Omron CX-Programmer project NewProject (CX-Programmer 9.66)

# PLC NewPLC1: CP1H XA

## Global symbols (name address type ; comment)
AI_SAW_CURRENT 200 CHANNEL  ; ANALOG.INPUT1.SAW.CURRENT
AI_TRANS_AXIS_DRIVE_VEL_FDBK 201 CHANNEL  ; AI.TRANSVERSE.AXIS.DRIVE.VELOCITY.FEEDBACK
AO_TRANS_VEL_REF 210 CHANNEL  ; TRANSVERSE.AXIS.VELOCITY.ANALOG.REFERENCE
0.05 BOOL  ; SPARE - Possible Zone Interference Limit Switch Input.
1024 CHANNEL  ; Encoder PPR
1.03 BOOL  ; Spare
200 CHANNEL  ; Saw Motor Current Input
210 CHANNEL  ; Cross Travel Speed Refernce Command
40 CHANNEL  ; OI.SCALING.SAW.CURRENT.PART1
8.00 BOOL  ; Place holder for Automatic PID control request
A434.04 BOOL  ; Analog IO Initialised
D100 CHANNEL  ; M_BLOCK_HEIGHT_INT_RAW
D10000 CHANNEL  ; OPERATION.PROGRAM.CHECK.BLOCK1.BLOCK.HEIGHT
D10001 CHANNEL  ; OPERATION.CHECK.PROGRAM.BLOCK1.BLOCK.QUANTITY
D10002 CHANNEL  ; OPERATION.PROGRAM.CHECK.BLOCK1.FORWARD.POSITION
D10003 CHANNEL  ; OPERATION.PROGRAM.CHECK.BLOCK1.FIRST.CUT
D10004 CHANNEL  ; OPERATION.PROGRAM.CHECK.BLOCK1.NUMBER.OF.SLABS
D10006 CHANNEL  ; OPERATION.PROGRAM.CHECK.BLOCK1.SLAB1.QUANTITY
D10007 CHANNEL  ; OPERATION.PROGRAM.CHECK.BLOCK1.SLAB2.SIZE
D10008 CHANNEL  ; OPERATION.PROGRAM.CHECK.BLOCK1.SLAB2.QUANTITY
D10009 CHANNEL  ; OPERATION.PROGRAM.CHECK.BLOCK1.SLAB3.SIZE
D1001 CHANNEL  ; Block 1 Data - Number of Blocks
D10010 CHANNEL  ; OPERATION.PROGRAM.CHECK.BLOCK1.SLAB1.SIZE
D10010 CHANNEL  ; OPERATION.PROGRAM.CHECK.BLOCK1.SLAB1.SIZE
D10011 CHANNEL  ; OPERATION.PROGRAM.CHECK.BLOCK1.SLAB4.SIZE
D10012 CHANNEL  ; OPEARTION.PROGRAM.CHECK.BLOCK1SLAB2.SIZE
D10013 CHANNEL  ; OPERATION.PROGRAM.CHECK.BLOCK1.SLAB5.SIZE
D10014 CHANNEL  ; OPERATION.PROGRAM.CHECK.BLOCK1.SLAB3.SIZE
D10016 CHANNEL  ; OPERATION.PROGRAM.CHECK.BLOCK1.SLAB4.SIZE
D10017 CHANNEL  ; OPERATION.PROGRAM.CHECK.BLOCK2.FORWARD.POSITION
D10018 CHANNEL  ; OPERATION.PROGRAM.CHECK.BLOCK1.SLAB5.SIZE
D10019 CHANNEL  ; OPERATION.PROGRAM.CHECK.BLOCK2.NUMBER.OF.SLABS
D10021 CHANNEL  ; OPERATION.PROGRAM.CHECK.BLOCK2.SLAB1.QUANTITY
D10023 CHANNEL  ; OPERATION.PROGRAM.CHECK.BLOCK2.SLAB2.QUANTITY
D10025 CHANNEL  ; OPERATION.PROGRAM.CHECK.BLOCK2.SLAB3.QUANTITY
D10027 CHANNEL  ; OPERATION.PROGRAM.CHECK.BLOCK2.SLAB4.QUANTITY
D10029 CHANNEL  ; OPERATION.PROGRAM.CHECK.BLOCK.2.SLAB5.QUANTITY
D101 CHANNEL  ; M_STORED.NUMBER_OF_BLOCKS
D10100 CHANNEL  ; OPERATION.PROGRAM.CHECK.BLOCK2.BLOCK.HEIGHT
D10120 CHANNEL  ; OPERATION.PROGRAM.CHECK.BLOCK2.SLAB1.SIZE
D10122 CHANNEL  ; OPERATION.PROGRAM.CHECK.BLOCK2.SLAB2.SIZE
D10124 CHANNEL  ; OPERATION.PROGRAM.CHECK.BLOCK2.SLAB3.SIZE
D10126 CHANNEL  ; OPERATION.PROGRAM.CHECK.BLOCK2.SLAB4.SIZE
D10128 CHANNEL  ; OPERATION.PROGRAM.CHECK.BLOCK2.SLAB5.SIZE
D10150 CHANNEL  ; OPERATION.PROGRAM.CHECK.BLOCK3.HEIGHT
D10160 CHANNEL  ; OPERATION.PROGRAM.CHECK.BLOCK3.SLAB1.SIZE
D10162 CHANNEL  ; OPERATION.PROGRAM.CHECK.BLOCK3.SLAB2.SIZE
D110 CHANNEL  ; Stored Block Height Float
D112 CHANNEL  ; Stored Target Position for Vertical Axis
D122 CHANNEL  ; OPERATION.SAW.CURRENT.INTERNAL
D2002 CHANNEL  ; OPERATION.PROGRAM.CHECK.BLOCK1.SLAB2.SIZE
D3000 CHANNEL  ; Input Data Table Control Word
D3001 CHANNEL  ; Maximum Anaolg Input Value (Xm)
D3002 CHANNEL  ; Y0
D3003 CHANNEL  ; X1
D3004 CHANNEL  ; Maximum Output value
D3100 CHANNEL  ; Output Data Control Word
D3101 CHANNEL  ; Xm
D3102 CHANNEL  ; Y0
D3103 CHANNEL  ; X1
D3104 CHANNEL  ; Y1
D32 CHANNEL  ; OPERATION.AUTO.CYCLE.BLOCK.FIRST.CUT.WORKING.REAL
D3200 CHANNEL  ; Setpoint Input Data Table Control Word
D3201 CHANNEL  ; Maximum Input Setpoint
D3202 CHANNEL  ; Y0
D3203 CHANNEL  ; X1
D3204 CHANNEL  ; Y1
D34 CHANNEL  ; OP.CONTROL.VERTICAL.TARGET.SCALED
D3520 CHANNEL  ; PID Setpoint Scaled for PID
D3521 CHANNEL  ; PID Instruction Proportional Component
D3522 CHANNEL  ; PID Instruction Integral Component
D3523 CHANNEL  ; PID Instruction Derivative Component
D3524 CHANNEL  ; PID Instruction Period
D3525 CHANNEL  ; PID Instruction Control Word
D3526 CHANNEL  ; PID Instruction Input and Output Range Setting
D3527 CHANNEL  ; PID Instruction Output Minimum
D3528 CHANNEL  ; PID Instruction Output Maximum
D36 CHANNEL  ; OPERATION.AUTO.CYCLE.VERTICAL.HIGH/LOW/SPEED.SELECT
D40 CHANNEL  ; OP.CONTROL.CURRENT.BLOCK.HEIGHT.REAL
D400 CHANNEL  ; Working Floating Point First Cut Value Current Block
D4000 CHANNEL  ; OPERATION.AUTO.CYCLE.BLK.PTR
D4002 CHANNEL  ; OPERATION.AUTO.CYCLE.BLOCK.DATA.POINTER
D4004 CHANNEL  ; OPERATION.CURRENT.PROGRAM.SLAB.DATA.POINTER
D4006 CHANNEL  ; OPERATION.AUTO.CYCLE.SPARE
D4008 CHANNEL  ; OPERATION.AUTO.CYCLE.SPARE
D4010 CHANNEL  ; OPERATION.SLAB.POINTER.THIS.BLOCK
D4012 CHANNEL  ; D4103
D4014 CHANNEL  ; OPERATION.AUTO.CYCLE.SLAB.POINTER
D42 CHANNEL  ; OP.CONTROL.CURRENT.BLOCK.LENGTH
D44 CHANNEL  ; OP.CONTROL.AUTO.CYCLE.VERTICAL.TARGET
D46 CHANNEL  ; OP.CONTROL.AUTO.TRANSVERSE.TARGET.FORWARD
D48 CHANNEL  ; OP.CONTROL.TRANSVERSE.POSITION.TARGET.REAL
D480 CHANNEL  ; Ctl.PID.Output.Value
D484 CHANNEL  ; Saw Current Scaled for PID instruction use
D50 CHANNEL  ; OPERATION.AUTO.CYCLE.BLOCK.HEIGHT.REAL
D500 CHANNEL  ; First Cut Position Stored Float
D502 CHANNEL  ; Stored Slab Size Inches Float
D504 CHANNEL  ; Total Slab Size Float
D506 CHANNEL  ; Stored Kerf Size Total
D508 CHANNEL  ; Slab Total Size Calc'd
D510 CHANNEL  ; Total of First Cut Position and Slab Size
D512 CHANNEL  ; Final Calculated Position at Cut Finish of this Slab and this Block
D52 CHANNEL  ; OPERATION.AUTO.CYCLE.BLOCK.TRANSVERSE.AXIS.FORWARD.STOP.POSITION
D54 CHANNEL  ; OPERATION.AUTO.CYCLE.BLOCK.FIRST.CUT.REAL
D5400 CHANNEL  ; OPERATION.LONG.TRAVEL.TARGET.WINDOW.PLUS
D5402 CHANNEL  ; OPERATION.LONG.TRAVEL.TARGET.WINDOW.MINUS
D5404 CHANNEL  ; OPERATION.LONG.TRAVEL.TARGET.WINDOW.SLABCUT.PLUS
D5406 CHANNEL  ; OPERATION.LONG.TRAVEL.TARGET.SLABCUT.MINUS
D5500 CHANNEL  ; OPERATION.AUTO.CYCLE.BLOCK.FIRST.CUT.REAL.SCALED
D5502 CHANNEL  ; OPERATION.AUTO.CYCLE.LON.INDEX.LOCATION.REAL.SCALED
D56 CHANNEL  ; OPERATION.AUTO.CYCLE.LONG.TARGET.KERF
D5600 CHANNEL  ; MC.TRANSVERSE.AXIS.POSITION.FEEDBACK.GB.SCALED.REAL
D58 CHANNEL  ; OPERATION.AUTO.CYCLE.ADD.KERF.TO.LOCATION.REAL
D6 CHANNEL  ; OPERATION.TRANSVERSE.AXIS.JOG.VELOCITY.REFERNCE.WORD
D60 CHANNEL  ; OPERATION.AUTO.CYCLE.LONG.INDEX.LOCATION.REAL
D6000 CHANNEL  ; MC.TRANSVERSE.AXIS.POSITION.FEEDBACK.RAW.REAL
D6002 CHANNEL  ; MC.TRANSVERSE.AXIS.POSITION.FEEDBACK.GB.SCALED.REAL
D6004 CHANNEL  ; MC.TRANSVERSE.AXIS.POSITION.PINION.REVOLUTIONS.REAL
D6006 CHANNEL  ; PI.EQUATION.PART.ONE
D6008 CHANNEL  ; PI.EQUATION.PART.TWO
D6012 CHANNEL  ; PI
D6014 CHANNEL  ; MC.TRANSVERSE.AXIS.PINION.CIRCUMFERENCE.INCHES.REAL
D66 CHANNEL  ; OPERATION.AUTO.CYCLE.CURRENT.SLAB.SIZE.REAL.RAW
D76 CHANNEL  ; OP.TRANSVERSE.AXIS.FORWARD.TARGET
D80 CHANNEL  ; Blade Kerf Raw Converted
D82 CHANNEL  ; Cut Depth Raw Converted
D84 CHANNEL  ; Cut Target Current Raw Converted
D86 CHANNEL  ; Current Slab Size Raw Converted
D97 CHANNEL  ; OP.CONTROL.AUTO.CYCLE.CURRENT.FIRST.CUT.LOCATION.LONG
D990 CHANNEL  ; PID Setpoint
H0.11 BOOL  ; OPERATION.ALARM.RESET.COMMAND
H10.13 BOOL  ; MC.LONG.AXIS.HOME.TIME.MON
H11.03 BOOL  ; VERTICAL.AXIS.DRIVE.NOT.OKAY
H11.07 BOOL  ; MC.VERTICAL.AXIS.JOG.PLUS
H11.08 BOOL  ; MC.VERTICAL.AXIS.JOG.MINUS
H11.13 BOOL  ; MC.VERTICAL.AXIS.DRIVE.RESET.ENABLED
H12.07 BOOL  ; MC.TRANSVERSE.AXIS.JOG.PLUS.INT
H12.08 BOOL  ; MC.TRANSVERSE.AXIS.JOG.NEG
H12.13 BOOL  ; MC.TRANSVERSE.AXIS.DRIVE.RESET.ENABLED
H13.04 BOOL  ; SAW.AUTO.RUN.UP.TIMER.DONE
H13.05 BOOL  ; OPERATION.AUTO.CYCLE.SAW.OVERCURRENT.ALARM
H13.06 BOOL  ; OPERATION.SAW.CURRENT.SENSING.CHECK.FAULT
H13.07 BOOL  ; OPERATION.SAW.MACHINE.STOP.COMMAND.ACTIVE
H13.08 BOOL  ; OPERATION.SAW.MACHINE.STOP.COMMAND.NOT ACTIVE
H13.15 BOOL  ; OP.ALARM.SAW.SOFT.START.FAULTED
H14.02 BOOL  ; WATER.FLOW.SHOULD.BE.ON
H14.03 BOOL  ; WATER.FLOW.IS.ON.AND.SHOULDN'T
H14.07 BOOL  ; OP.WATER.MACHINE.STOP.COMMAND.ACTIVE
H14.08 BOOL  ; OP.WATER.MACHINE.sTOP.COMMAND.NOT.ACTIVE
H14.14 BOOL  ; OP.ALARM.WATER.FLOW.ERROR
H16.14 BOOL  ; RECIPE.ERROR
H1.00 BOOL  ; OP.MODE.INDICATOR.ENABLED
H1.01 BOOL  ; OP.MODE.AUTO.PGM.CHECK.ACT
H1.02 BOOL  ; OP.MODE.AUTO.PGM.CHECK.CMP
H1.03 BOOL  ; LAST.BLOCK.CHECK
H1.14 BOOL  ; ALARM.RESEST.TRAP
H1.15 BOOL  ; MODE.AUTO.GATE.ALARM.TRIGGER
H2 CHANNEL  ; Cycle Start Bits
H20.04 BOOL  ; Data Convert Done
H20.05 BOOL  ; OPERATION.SET.FIRST.CUT.LOCATION.LONG.TARGET
H20.06 BOOL  ; OP.CONTROL.AUTO.CYCLE.INDEX.LONG.AXIS
H20.07 BOOL  ; OPERATION.AUTO.CYCLE.LONG.AXIS.INDEX.COMMAND.SYNC
H20.08 BOOL  ; OPERATION.LONG.AXIS.IN.POSITION.WINDOW.TOLERANCE
H20.09 BOOL  ; OPERATION.AUTO.CYCLE.LONG.AXIS.SLAB.TARGET.CALCED
H20.12 BOOL  ; OP.LONG.AXIS.MACHINE.STOP.ACTIVE
H20.13 BOOL  ; OP.LON.AXIS.MACHINE.STOP.NOT.ACTIVE
H20.14 BOOL  ; OP.CONTROL.INTERLOCK.LONG.AXIS.IN.MOTION
H21.05 BOOL  ; MC.VERTICAL.AXIS.HOME.INIT
H21.08 BOOL  ; OP.CONTROL.VERTICAL.IN.POSITION
H21.09 BOOL  ; OP.CONTROL.VERTICAL.HIGH.SPEED.SELECT
H21.10 BOOL  ; OP.CONTROL.VERTICAL.TARGET.CALC
H21.12 BOOL  ; OP.VERTICAL.AAXIS.MACHINE.STOP.ACTIVE
H21.13 BOOL  ; OP.VERTICAL.AXIS.MACHINE.STOP.NOT.ACTIVE
H21.14 BOOL  ; OP.CONTROL.INTERLOCK.VERTICAL.AXIS.IN.MOTION
H22.05 BOOL  ; MC.TRANSVERSE.AXIS.HOMING.REQUEST
H22.06 BOOL  ; OPERATION.AUTO.TRANSVERSE.AXIS.IN.FORWARD.POSITION
H22.07 BOOL  ; OP.TRANSVERSE.DIRECTION.DISCRIMINATOR
H22.08 BOOL  ; OP.CONTROL.AUTO.CYCLE.TRANSVERSE.AXIS.MOTION.ENABLE
H22.09 BOOL  ; OP.AUTO.CYCLE.TRANSVERS.AXIS.NOT.IN.POSITION.FORWARD
H22.10 BOOL  ; OP.CONTROL.TRANSVERSE.TARGET.CALC
H22.12 BOOL  ; OP.TRANSVERSE.AXIS.MACHINE.STOP.ACTIVE
H22.13 BOOL  ; OP.TRANSVERSE.AXIS.MACHINE.STOP.NOT.ACTIVE
H22.14 BOOL  ; OP.CONTROL.INTERLOCK.TRANS.AXIS.IN.MOTION
H2.00 BOOL  ; CYCLE.START.ENABLE
H2.01 BOOL  ; CYCLE.START.FUNCTION.RESET
H2.02 BOOL  ; CYCLE.START.FUNCTION.ENABLED
H2.03 BOOL  ; CYCLE.START.ACTIVE
H2.04 BOOL  ; CYCLE.START.COMPLETE
H2.05 BOOL  ; OPERATION.AUTO.CYCLE.START.COMMAND
H2.14 BOOL  ; CYCLE.START.ERROR
H32.07 BOOL  ; OPERATION.PROGRAM.CHECK.BLOCK1.ENABLE
H32.08 BOOL  ; OPERATION.PROGRAM.CHECK.BLOCK1.ENABLE
H32.09 BOOL  ; OPERATION.PROGRAM.CHECK.BLOCK2.ENABLE
H32.10 BOOL  ; OPERATION.PROGRAM.CHECK.BLOCK3.ENABLE
H35.00 BOOL  ; OPERATION.PROGRAM.CHECK.BLOCK1.ENABLE
H3.00 BOOL  ; OP_CTL_CYCLE_RUN_ENABLE
H3.01 BOOL  ; OP.CONTROL.CYCLE.RUN.ENABLED
H3.02 BOOL  ; CYCLE.RUN.ACTIVE
H3.03 BOOL  ; MACHINE.CYCLE.STOP
H3.04 BOOL  ; CYCLE.STOP.COMMAND
H3.05 BOOL  ; OPERATION.AUTO.CYCLE.STOP.COMMAND
H3.06 BOOL  ; OPERATION.CYCLE.RUN.RESET
H3.14 BOOL  ; CYCLE.RUN.ERROR
H4 CHANNEL  ; Cycle Stop Bits
H4.00 BOOL  ; CYCLE.STOP.ENABLE
H4.01 BOOL  ; CYCLE.STOP.INSTRUCTION.RESET
H4.02 BOOL  ; CYCLE.STOP.FUNCTION.ENABLE
H4.03 BOOL  ; CYCLE.STOP.ACTIVE
H4.04 BOOL  ; CYCLE.STOP.COMPLETE
H4.05 BOOL  ; OPERATION.AUTO.CYCLE.ISSUE.SAFE.TO.STOP.COMMAND
H4.08 BOOL  ; OPERTION.CYCLE.STOP.COMMAND.INITIATED
H4.14 BOOL  ; CYCLE.STOP.INSTRUCTION.ERROR
H5.03 BOOL  ; GLOBAL.HOME.REQUEST.ACTIVE
H7 CHANNEL  ; Auto Cycle Step Word 1
H7.00 BOOL  ; OPERATION.AUTO.CYCLE.SEQUENCE.STEP1
H7.01 BOOL  ; OPERATION.AUTO.CYCLE.SEQUENCE.STEP2
H7.02 BOOL  ; OPERATION.AUTO.CYCLE.SEQUENCE.STEP3
H7.03 BOOL  ; OPERATION.AUTO.CYCLE.SEQUENCE.STEP4
H7.04 BOOL  ; OPERATION.AUTO.CYCLE.SEQUENCE.STEP5
H7.05 BOOL  ; OPERATION.AUTO.CYCLE.SEQUENCE.STEP6
H7.06 BOOL  ; OPERATION.AUTO.CYCLE.SEQUENCE.STEP7
H7.07 BOOL  ; OPERATION.AUTO.CYCLE.SEQUENCE.STEP8
H7.08 BOOL  ; OPERATION.AUTO.CYCLE.SEQUENCE.STEP9
H7.09 BOOL  ; OPERATION.AUTO.CYCLE.SEQUENCE.STEP10
H7.10 BOOL  ; OPERATION.AUTO.CYCLE.SEQUENCE.STEP11
H7.11 BOOL  ; OPERATION.AUTO.CYCLE.SEQUENCE.STEP12
H7.12 BOOL  ; OPERATION.AUTO.CYCLE.SEQUENCE.STEP13
H7.13 BOOL  ; OPERATION.AUTO.CYCLE.SEQUENCE.STEP14
H7.14 BOOL  ; OPERATION.AUTO.CYCLE.SEQUENCE.STEP15
H7.15 BOOL  ; OPERATION.AUTO.CYCLE.SEQUENCE.STEP16
H8 CHANNEL  ; Auto Cycle Step Word 2
H8.00 BOOL  ; OPERATION.AUTO.CYCLE.SEQUENCE.STEP17
H8.01 BOOL  ; OPERATION.AUTO.CYCLE.SEQUENCE.STEP18
H8.02 BOOL  ; OPERATION.AUTO.CYCLE.SEQUENCE.STEP19
H8.03 BOOL  ; OPERATION.AUTO.CYCLESEQUENCE.STEP20
H8.04 BOOL  ; OPERATION.AUTO.CYCLE.SEQUENCE.STEP21
H8.05 BOOL  ; OPERATION.AUTO.CYCLE.SEQUENCE.STEP22
H8.06 BOOL  ; OPERATION.AUTO.CYCLE.SEQUENCE.STEP23
H8.07 BOOL  ; OPERATION.AUTO.CYCLE.SEQUENCE.STEP24
H8.08 BOOL  ; OPERATION.AUTO.CYCLESEQUENCE.STEP25
H8.09 BOOL  ; OPERATION.AUTO.CYCLE.SEQUENCE.STEP26
H8.10 BOOL  ; OPERATION.AUTO.CYCLE.SEQUENCE.STEP27
H9 CHANNEL  ; OPERATION.AUTO.CYCLE.SEQUENCE.STATE.BITS
H9.00 BOOL  ; OPERATION.AUTO.CYCLE.FIRST.CUT.COMPLETED
H9.01 BOOL  ; OPERATION.AUTO.CYCLE.BLOCK.COMPLETE
H9.02 BOOL  ; OPERATION.AUTO.CYCLE.CURRENT.BLOCK.NO.SLABS.BIT
H9.03 BOOL  ; OPERATION.AUTO.CYCLE.ZERO.HEGHTBLOCK
H9.15 BOOL  ; OPERATION.AUTO.CYCLE.STEP.ENABLE
T0000 BOOL  ; Step 0 Timer Done
T0001 BOOL  ; Step 1 Timer Done
T0002 BOOL  ; Step 2 timer done
T0003 BOOL  ; Increment Slab Pulse Timer
T0004 BOOL  ; Slab Decrement Pulse Timer
T0005 BOOL  ; Block Increment Pulse Timer
T0006 BOOL  ; Block Decrement Pulse Timer
T0010 BOOL  ; Block Step 0 Timer
T0011 BOOL  ; Block Step 1 Timer
T0012 BOOL  ; Block Step 2 Timer
T0013 BOOL  ; Block Step 3 Timer
T0014 BOOL  ; Block Step 4 timer
T0015 BOOL  ; Block Step 5 Timer
T0016 BOOL  ; Block Step 6 Timer
T0017 BOOL  ; Saw Current At Limit Timer
T0018 BOOL  ; OPERATION.SAW.CURRENT.SENSING.ZERO.CURRENT.CHECK.TIMER
T0020 BOOL  ; MC.VERTICAL.AXIS.BRAKE.TIMER
T0021 BOOL  ; MC.LONG.AXIS.HOME.ACT.TIMER
T0022 BOOL  ; MC.LONG.AXIS.INDEX.COMMAND.COMPLETE.TIME
T0023 BOOL  ; Index Position Data Setle Timer
T0029 BOOL  ; OPERATION.AUTO.CYCLE.SEQUENCE.STEP1.TIMER
T0030 BOOL  ; OPERATION.AUTO.CYCLE.STEP2.TIMER
T0031 BOOL  ; OPERATION.SEQUENCE.STEP3.TIMER
T0032 BOOL  ; OPERATION.AUTO.CYCLE.SEQUENCE.STEP4.TIMER
T0033 BOOL  ; OPERATION.AUTO.CYCLE.SEQUENCE.STEP5.TIMER
T0034 BOOL  ; OPERATION.AUTO.CYCLE.SEQUENCE.STEP6.TIMER
T0035 BOOL  ; OPERATION.AUTO.CYCLE.SEQUENCE.STEP7.TIMER
T0036 BOOL  ; OPERATION.AUTO.CYCLE.SEQUENCE.STEP8.TIMER
T0037 BOOL  ; OPERATION.AUTO.CYCLE.SEQUENCE.STEP9.TIMER
T0038 BOOL  ; OPERATION.AUTO.CYCLE.SEQUENCE.STEP10.TIMER
T0039 BOOL  ; OPERATION.AUTO.CYCLE.SEQUENCE.STEP11.TIMER
T0040 BOOL  ; OPERATION.AUTO.CYCLE.SEQUENCE.STEP12.TIMER
T0041 BOOL  ; OPERATION.AUTO.CYCLE.SEQUENCE.STEP13.TIME
T0042 BOOL  ; OPERATION.AUTO.CYCLE.STEP14.TIMER
T0043 BOOL  ; OPERATION.AUTO.CYCLE.STEP15.TIMER
T0044 BOOL  ; OPERATION.AUTO.CYCLE.SEQUENCE.STEP16.TIMER
T0045 BOOL  ; OPERATION.AUTO.CYCLE.SEQUENCE.STEP17.TIMER
T0046 BOOL  ; OPERATION.AUTO.CYCLE.SEQUENCE.STEP18.TIMER
T0047 BOOL  ; OPERATION.AUTO.CYCLE.SEQUENCE.STEP19.TIMER
T0048 BOOL  ; OPERATION.AUTO.CYCLE.SEQUENCE.STEP20.TIMER
T0049 BOOL  ; OPERATION.AUTO.CYCLE.SEQUENCE.STEP21.TIMER
T0050 BOOL  ; OPERATION.AUTO.CYCLE.SEQUENCE.STEP22.TIMER
T0051 BOOL  ; OPERATION.AUTO.CYCLE.SEQUENCE.STEP23.TIMER
T0052 BOOL  ; OPERATION.AUTO.CYCLE.STEP24.TIMER
T0053 BOOL  ; OPERATION.AUTO.CYCLE.SEQUENCE.STEP25.TIMER
T0054 BOOL  ; OPERATION.AUTO.CYCLE.SEQUENCE.STEP26.TIMER
T0100 BOOL  ; Index Delay Time
T0101 BOOL  ; OPERATION.LONG.AXIS.INDEX.COMMAND.START.DELAY.TIMER
T0130 BOOL  ; OPERATION.AUTO.CYCLE.SAW.RUN.UP.TIME
T0200 BOOL  ; OPERATION.CONTROL.RESET.SEQUENCE.TIMER
W0.01 BOOL  ; Test Bit Blocker. Remove when done
W0.02 BOOL  ; W0.11
W0.12 BOOL  ; GLOBAL.HOME.REQUEST.HOME.TRANSVERSE
W0.13 BOOL  ; GLOBAL.HOME.REQUEST.HOME.VERTICAL
W0.14 BOOL  ; CTL.GLOBAL.HOME.REQUEST.COMPLETED
W102.00 BOOL  ; OI.MESSAGE.INTERNAL.TRIGGER.MSG1
W102.01 BOOL  ; OI.MESSAGE.MSG2.TRIGGER
W102.02 BOOL  ; OI.MESSAGE.MSG3.TRIGGER
W102.03 BOOL  ; OI.MESSAGE.MSG4.TRIGGER
W102.04 BOOL  ; OI.MESSAGE.MSG5.TRIGGER
W102.05 BOOL  ; OI.MESSAGE.MSG6.TRIGGER
W102.06 BOOL  ; OI.MESSAGE.MSG7.TRIGGER
W102.07 BOOL  ; OI.MESSAGE.MSG8.TRIGGER
W102.08 BOOL  ; OI.MESSAGE.MSG9.TRIGGER
W102.09 BOOL  ; OI.MESSAGE.MSG10.TRIGGER
W104.00 BOOL  ; OI.MESSAGES.ENABLED
W104.01 BOOL  ; OI.MESSAGE.MSG2.ENABLED
W104.15 BOOL  ; OI.GLOBAL.MESSAGE.TRIGGER
W105 CHANNEL  ; OI.MESSAGE.SELECTION.INTERNAL
W108 CHANNEL  ; OI.MESSAGE.COLOUR.INTERNAL
W109 CHANNEL  ; OI.MESSAGE.SELECT.INTERNAL
W112.00 BOOL  ; OI.ALARM.MESSAGE.MSG1.TRIGGER
W112.01 BOOL  ; OI.ALARM.MESSAGE.SELECT.MSG2.TRIGGER
W112.02 BOOL  ; OI.ALARM.MESSAGE.MSG3.TRIGGER
W112.03 BOOL  ; OI.ALARM.MESSAGE.MSG4.TRIGGER
W112.04 BOOL  ; OI.ALARM.MESSAGE.MSG5.TRIGGER
W112.05 BOOL  ; OI.ALARM.MESSAGE.MSG6.TRIGGER
W112.09 BOOL  ; OI.ALARM.MESSAGE.MSG10.TRIGGER
W112.10 BOOL  ; OI.ALARM.MESSAGE.MSG11.TRIGGER
W112.12 BOOL  ; OI.ALARM.MESSAGE.MSG13.TRIGGER
W112.13 BOOL  ; OI.ALARM.MESSAGE.MSG14.TRIGGER
W112.15 BOOL  ; OI.ALARM.MESSAGE.MSG16.TRIGGER
W113.05 BOOL  ; OI.ALARM.MESSAGE.MSG21.TRIGGER
W113.06 BOOL  ; OI.ALARM.MESSAGE.MSG22.TRIGGER
W113.07 BOOL  ; OI.ALARM.MESSAGE.MSG13.TRIGGER
W113.15 BOOL  ; OI.ALARM.MESSAGE.MSG31.TRIGGER
W114.00 BOOL  ; OI.ALARM.MESSAGE.MSG1.ENABLED
W114.01 BOOL  ; OI.ALARM.MESSAGE.MSG32.TRIGGER
W114.02 BOOL  ; OI.ALARM.MESSAGE.MSG33.TRIGGER
W114.03 BOOL  ; OI.ALARM,.MESSAGE.MSG34.TRIGGER
W114.15 BOOL  ; OI.ALARM.MESSAGE.TRIGGER.GLOBAL
W115 CHANNEL  ; OI.INTERNAL.ALARM.MESSAGE.SELECTION
W116.00 BOOL  ; OI.ALARM.MESSAGE.MSG51.TRIGGER
W116.01 BOOL  ; OI.ALARM.MESSAGE.MSG52.TRIGGER
W116.02 BOOL  ; OI.ALARM.MESSAGE.MSG53.TRIGGER
W116.03 BOOL  ; OI.ALARM.MESSAGE.MSG54.TRIGGER
W117.00 BOOL  ; OI.ALARM.MESSAGE.MSG71.TRIGGER
W117.01 BOOL  ; OI.ALARM.MESSAGE.MSG72.TRIGGER
W117.02 BOOL  ; OI.ALARM.MESSAGE.MSG73.TRIGGER
W117.03 BOOL  ; ALARM.MESSAGE.MSG74.TRIGGER
W117.04 BOOL  ; OI.ALARM.MESSAGE.MSG75.TRIGGER
W118 CHANNEL  ; OI.ALARM.MESSAGE.COLOUR.SELECT.INTERNAL
W120.09 BOOL  ; OI.VERTICAL.AXIS.HOME.REQUEST.PB
W121.02 BOOL  ; Previous Block
W121.03 BOOL  ; Previous Slab of Current Block
W121.04 BOOL  ; Next Slab of current Block
W121.05 BOOL  ; Next Block Select
W121.07 BOOL  ; Clear Data
W121.09 BOOL  ; OI.ALARM.ACCEPT.CONFIRMATION
W121.10 BOOL  ; OI.CONTROL.RESET.AUTO.CYCLE.SEQUENCE
W12.00 BOOL  ; Slab Change Data Storage and Display Update Step 0
W12.01 BOOL  ; Step 1
W12.02 BOOL  ; Step 2
W12.03 BOOL  ; Step 3
W12.04 BOOL  ; Step 4
W12.05 BOOL  ; Step 5
W12.06 BOOL  ; Step 6
W12.15 BOOL  ; Loop Step Reset
W130.00 BOOL  ; OI.ALL.HOME.INDICATOR
W130.04 BOOL  ; OI.VERTICAL.AXIS.HOME.INDICATOR
W130.05 BOOL  ; OI.VERTICAL.AXIS.JOG.FORWARD.INDICATOR
W130.06 BOOL  ; OI.VERTICAL.AXIS.JOG.REVERSE.INDICATOR
W130.07 BOOL  ; OI.INDICATE.TRANSVERSE.AXIS.HOME.INDICATOR
W130.08 BOOL  ; OI.TRANSVERSE.AXIS.JOG.REVERSE.INDICATOR
W130.09 BOOL  ; OI.TRANSVERSE.AXIS.JOG.FORWARD.INDICATOR
W130.10 BOOL  ; OI.LONG.AXIS.JOG.RIGHT.COMMAND.ACTIVE.INDICATOR
W130.11 BOOL  ; OI.LONG.AXIS.JOG.LEFT.COMMAND.ACTIVE.INDICATOR
W130.12 BOOL  ; OI.LONG.AXIS.HOME.INDICATOR
W131.00 BOOL  ; OI.SLAB.INCREMENT.PB.ENABLE
W131.01 BOOL  ; OI.BLOCK.POINTER.INCREMENT.PB.ENABLE
W13.00 BOOL  ; Step 0 in Progress
W13.01 BOOL  ; Step 1 in Progress
W13.02 BOOL  ; Step 2 in Progress
W13.03 BOOL  ; Step 3 in Progress
W13.04 BOOL  ; Step 4 in Progress
W13.05 BOOL  ; Step 5 in Progress
W13.06 BOOL  ; Step 6 in Progress
W14.00 BOOL  ; Step 0 Done
W14.01 BOOL  ; Step 1 Done
W14.02 BOOL  ; Step 2 Done
W14.03 BOOL  ; Step 3 Done
W14.04 BOOL  ; Step 4 Done
W14.05 BOOL  ; Step 5 Done
W14.06 BOOL  ; Step 6 Done
W150 CHANNEL  ; Block Number Captured
W151 CHANNEL  ; Number of Words for Blocks
W152 CHANNEL  ; Slab Count Work Word for Block Pointer
W153 CHANNEL  ; Offset Calculate for Last Slab Count
W154 CHANNEL  ; Offset Mid Calc
W156 CHANNEL  ; Offset Calc'd
W158 CHANNEL  ; Slab Record Offset Interim
W15.00 BOOL  ; Block Change Data Storage and Display Update Step 0
W15.01 BOOL  ; Loop Step 1
W15.02 BOOL  ; Loop Step 2
W15.03 BOOL  ; Loop Step 3
W15.04 BOOL  ; Loop Step 4
W15.05 BOOL  ; Loop Step 5
W15.06 BOOL  ; Loop Step 6
W15.15 BOOL  ; Loop Step Reset
W160 CHANNEL  ; Slab Offset Result
W16.00 BOOL  ; Step 0 in Progress
W16.01 BOOL  ; Loop Step 1 in Progress
W16.02 BOOL  ; Loop Step 2 in Progress
W16.03 BOOL  ; Loop Step 3 in Progress
W16.04 BOOL  ; Loop Step 4 in Progress
W16.05 BOOL  ; Loop Step 5 in Progress
W16.06 BOOL  ; Loop Step 6 in Progress
W16.10 BOOL  ; Slab Data Read in Progress
W16.11 BOOL  ; Block Data Read in Progress
W17.00 BOOL  ; Step 0 Done
W17.01 BOOL  ; Loop Step 1 Done
W17.02 BOOL  ; Loop Step 2 Complete
W17.03 BOOL  ; Loop Sstep 3 Complete
W17.04 BOOL  ; Loop Step 4 Complete
W17.05 BOOL  ; Loop Step 5 Complete
W17.06 BOOL  ; Loop Step 6 Complete
W190 CHANNEL  ; Slab Pointer Offset Adjustment
W191 CHANNEL  ; Block 1 Slab Count Capture
W192 CHANNEL  ; Slab Offset Addition for This Block
W193 CHANNEL  ; Slab_ID_Raw
W194 CHANNEL  ; Slab Pointer Calculated
W195 CHANNEL  ; Slab Offset Previous
W196 CHANNEL  ; Slab_Offset_Constant_Calculated
W197 CHANNEL  ; Block_Selected_Base
W198 CHANNEL  ; Block Pointer Offset Calculated
W19.00 BOOL  ; Test Bit
W19.01 BOOL  ; Self Toggle
W1.01 BOOL  ; Test Bit 2
W200 CHANNEL  ; Current Programming Block ID
W201 CHANNEL  ; Current Programming Number Of Blocks
W202 CHANNEL  ; Current Programming Block Height
W203 CHANNEL  ; Current Programming Block Number of Blocks
W204 CHANNEL  ; Current Programming Block Cross Stop Location
W205 CHANNEL  ; Current Programming Block First Cut Location
W206 CHANNEL  ; Current Block Programmed Slab Count
W207 CHANNEL  ; Current Programming Slab ID
W208 CHANNEL  ; Current Slab Programmed Size in inches
W209 CHANNEL  ; Current Slab Programmed Quantity to cut
W20.00 BOOL  ; Block Incremented Pulse - Lead
W20.01 BOOL  ; Block Decremented Pulse - Lead
W20.02 BOOL  ; Slab Incremented Pulse - Lead
W20.03 BOOL  ; Slab Decremented Pulse - Lead
W20.04 BOOL  ; Slab Count Capture Trap
W20.05 BOOL  ; Block Read In Progress
W20.06 BOOL  ; Slab Count Changed from Block Read
W20.07 BOOL  ; Slab Pointer Updating
W20.08 BOOL  ; Update Working Offset
W20.09 BOOL  ; Block Pointer Calculate Enable
W20.10 BOOL  ; Increment Block Pointer
W20.11 BOOL  ; Decrement Block Pointer
W20.12 BOOL  ; First_Pass_Read
W20.14 BOOL  ; Block Offset Calculated
W20.15 BOOL  ; Block Program Control Enabled
W21.00 BOOL  ; Blade Kerf Data Write to Storage
W21.01 BOOL  ; Blade Kerf Read from Storage
W21.02 BOOL  ; Cut Depth Write to Storage
W21.03 BOOL  ; Cut Depth Read from Storage
W21.04 BOOL  ; Target Saw Current in Amps Write to Storage
W21.05 BOOL  ; Target Saw Current in Amps Read from Storage
W21.06 BOOL  ; Read Slab Data from Storage
W21.07 BOOL  ; Block Data Write to Storage
W21.08 BOOL  ; Automatic Number of Blocks Update
W21.09 BOOL  ; Slab Pointer Control Enabled
W21.10 BOOL  ; Increment Slab Offset
W21.11 BOOL  ; Decrement Slab Offset
W21.12 BOOL  ; Automatic Number of Slabs Update
W21.13 BOOL  ; Slab Pointer Reset
W21.14 BOOL  ; Block Pointer Reset
W22.00 BOOL  ; Slab Pointer Calculated
W22.01 BOOL  ; Block Pointer Changed
W22.02 BOOL  ; Current Block Selected Changed Initiate Block Data Write
W22.03 BOOL  ; Block Data Write Step Zero Complete
W22.04 BOOL  ; Block Data Write Complete
W22.05 BOOL  ; Capture Current Slab Words
W22.06 BOOL  ; Slab Data Write In Progress
W22.07 BOOL  ; Slab Data Write Complete
W22.08 BOOL  ; Block Offset Adjusted
W22.09 BOOL  ; Block Offset Adjust Complete
W22.10 BOOL  ; Block Data Read in Progress
W22.11 BOOL  ; Block Data Read >
W22.12 BOOL  ; Block Data Read Complete
W22.13 BOOL  ; Slab Offset Adjust in Progress
W22.14 BOOL  ; Slab Offset Adjust >
W22.15 BOOL  ; Slab Offset Adjust Complete
W23.00 BOOL  ; Slab Offset Init
W23.01 BOOL  ; Slab Offset Pointer Updating
W23.02 BOOL  ; Slab Offset Updated
W23.03 BOOL  ; Slab Data Read in Progress
W23.04 BOOL  ; Slab Data Read >
W23.05 BOOL  ; Slab Data Read Complete
W23.15 BOOL  ; Slab Offset Init Complete
W24.01 BOOL  ; Offset Init Step 1 Complete
W24.02 BOOL  ; OffsetInit Step 2 Complete
W24.03 BOOL  ; Offset Init Step 3 Complete
W250 CHANNEL  ; Offset value for Second word in indirect addressed storage area for Block Start Edge
W251 CHANNEL  ; Offset Value for Third word in Storge area for block length
W252 CHANNEL  ; Offset value calculated for 4th word in Storage area for block First Cut
W253 CHANNEL  ; Offset value calculated for number of slabs for current block
W256 CHANNEL  ; Last Slab Count from First Block
W257 CHANNEL  ; Offset adjust
W25.01 BOOL  ; Offset Init Step 1 In Progress
W25.02 BOOL  ; Offset Init Step 2 In Progress
W25.03 BOOL  ; Offset Init Step 3 In Progress
W26.00 BOOL  ; Minus Slab Offset Init
W26.01 BOOL  ; Minus Offset Init Step 1
W26.02 BOOL  ; Minus Offset Init Step 2
W26.03 BOOL  ; Minus Offset Init Step 3
W26.15 BOOL  ; Minus Slab Offset Init Complete
W27.01 BOOL  ; Minus Offset Init Step 1 Complete
W27.02 BOOL  ; Minus Offset Init Step 2 Complete
W27.03 BOOL  ; Minus Offset Init Step 3 Complete
W28.01 BOOL  ; Minus Offset Init Step 1 In Progress
W28.02 BOOL  ; Minus Offset Init Step 2 In Progress
W28.03 BOOL  ; Minus Offset Init Step 3 In Progress
W2.00 BOOL  ; Program Check - Increment Slab Pointer
W2.01 BOOL  ; Program Check - Increment Block
W2.02 BOOL  ; Program Check - Completed
W2.05 BOOL  ; Reset Pointer after Program Check
W300 CHANNEL  ; Blade Kerf Working
W301 CHANNEL  ; Cut Depth Working
W302 CHANNEL  ; Target Current Working
W30.00 BOOL  ; OI.MESSAGE.INTERNAL.TRIGGER.MSG1
W30.01 BOOL  ; OI.MESSAGE.INTERNAL.TRIGGER.MSG2
W30.09 BOOL  ; OI.ALARM.MESSAGE.TRIGGER.MSG10
W312 CHANNEL  ; Last Height Value for Current Block
W313 CHANNEL  ; Current Block Stored Height Data
W314 CHANNEL  ; Curren Block Number of Blocks
W315 CHANNEL  ; Current Block Stored Number of Blocks
W316 CHANNEL  ; Current Block Last Cross Stop Location
W317 CHANNEL  ; Current Block Stored Cross Stop Location
W318 CHANNEL  ; Current Block Last First Cut Position
W319 CHANNEL  ; Current Block Stored First Cut Location
W31.00 BOOL  ; OI.MESSAGE.CONTROL.ENABLED
W320 CHANNEL  ; Current Block Last Number of Slabs
W321 CHANNEL  ; Current Block Stored Slab Count
W322 CHANNEL  ; Current Slab Last Width
W323 CHANNEL  ; Current Slab Stored Width
W324 CHANNEL  ; Current Slab Last Quantity
W325 CHANNEL  ; Current Slab Stored Quantity
W350 CHANNEL  ; Axis position display
W37.00 BOOL  ; Current Height and Last Height are not Equal after Block Inc/Dec
W37.01 BOOL  ; Last Height and Stored Height are not Equal
W37.02 BOOL  ; Current Block Number of Blocks and Las Block Number of Blocks are Not Equal
W37.03 BOOL  ; Last Block Number of Blocks and Stored Value are not equal
W37.04 BOOL  ; Current Block Cross Stop Locations and Last Block Cross Stop Location are not equal
W37.05 BOOL  ; Last Block Cross Stop Location and Stored Cross Stop Location are Not Equal
W37.06 BOOL  ; Current and Last First Cut Location are Not Equal
W37.07 BOOL  ; Last and Stored First Cut Location are Not Equal
W37.08 BOOL  ; Last and Current Slab Count are Not Equal
W37.09 BOOL  ; Last and Stored Slab Count are Not Equal
W37.10 BOOL  ; Current and Last Slab Size are Not Equal
W37.11 BOOL  ; Last and Stored Slab Sizes are Not Equal
W37.12 BOOL  ; Last and Current Slab Qty are Not Equal
W37.13 BOOL  ; Last and Stored Slab Qty are Not Equal
W3.00 BOOL  ; STEP.ONE.EXECUTE
W3.01 BOOL  ; STEP.TWO.EXECUTE
W3.02 BOOL  ; STEP.THREE.EXECUTE
W400 CHANNEL  ; Temporary Storage for Block Data Used in Slab Offset Calc
W400.00 BOOL  ; Data Write Step
W400.01 BOOL  ; Data Offset Adjust Step
W400.02 BOOL  ; Data Read Step
W400.03 BOOL  ; End Step
W404 CHANNEL  ; # of Slabs for current Block
W405 CHANNEL  ; Number of words used by slabs in this block
W406 CHANNEL  ; Temporary Offset Storage word
W40.00 BOOL  ; Data Write/Read Sequence Initiate
W40.01 BOOL  ; Data Write Step Action
W40.02 BOOL  ; Data Offset Adjust Action
W40.03 BOOL  ; Data Read Step Action
W41.00 BOOL  ; Slab Data Write in Progress
W41.01 BOOL  ; Slab Data Write >
W41.02 BOOL  ; Slab Offset Adjust in Progress
W41.03 BOOL  ; Calulating Number of Words to Read
W4.00 BOOL  ; Program Check - Block First Cut Error
W4.01 BOOL  ; Program Check Step 1 - Block Pointer Reset
W4.02 BOOL  ; Program Check Step 1 - Ready for Next Step
W4.03 BOOL  ; Program Check Step 1 _ Store First Cut Position as Floating Point
W4.04 BOOL  ; Program Check Step 2 - Calculation Settle
W4.05 BOOL  ; Program Check Step 3 - Slab Size Convert to Floating Point
W4.06 BOOL  ; Program Check Step 3 - Totalise Kerf and Slab sizes Claculate Slab Size
W4.07 BOOL  ; Slab Size Calc
W4.08 BOOL  ; Calculate Kerf Total
W4.09 BOOL  ; Program Check Step 3 - Kerf Total Calculation
W4.10 BOOL  ; Program Check Step 3 - Add Kerf Total to Slab Size Total
W4.11 BOOL  ; Program Check Step 3 - Total Size Calculation => Position Target
W4.12 BOOL  ; Program Check Step 3 - Slab Inrement
W4.13 BOOL  ; Program Check Step 3 - Phase 2
W4.15 BOOL  ; Program Check Step 3 - Ready for Next Step
W5.00 BOOL  ; GLOBAL.HOME.REQUEST.HOME.LONG.TRAVEL
W5.01 BOOL  ; OPERATION.AUTO.CYCLE.SLAB.POINTER.INCREMENTED
W6.04 BOOL  ; OP.CONTROL.AUTO.CYCLE.RUN.EXECUTE.STEP2
W6.05 BOOL  ; OP.CONTROL.AUTO.CYCLE.RUN.STEP2
W6.06 BOOL  ; OP.CONTROL.AUTO.CYCLE.STEP3.RUN
W6.07 BOOL  ; OP.CONTROL.AUTO.CYCLE.RUN.STEP3.RAISE.VERTICAL
W6.08 BOOL  ; OP.CONTROL.RAISE.VERTICAL
W6.09 BOOL  ; OP.CONTROL.AUTO.CYCLE.STEP4
W6.10 BOOL  ; OP.CONTROL.AUTO.CYCLE.RUN.STEP4.INDEX.LONG
W7.00 BOOL  ; AUTO.MODE.ENABLED.RESET.WORKING.TO.FIRST.BLOCK
W7.03 BOOL  ; AUTO.SEQUENCE.STEP4.DN
W7.04 BOOL  ; Ctl.PID.Executing
W7.05 BOOL  ; Ctl.PID.Error
W7.06 BOOL  ; Current Position is Desired Position
W7.07 BOOL  ; MC.LONG.AXIS.INDEX.COMMAND.ACTIVE
W7.08 BOOL  ; MC.LONG.AXIS.INDEX.COMMAND.COMPLETED
W7.09 BOOL  ; OP.CONTROL.AUTO.CYCLE.RUN.SAW.MOTION
W7.10 BOOL  ; OP.CONTROL.INDEX.LONG
W8.00 BOOL  ; Place holder for auto index action Testing
W8.01 BOOL  ; OPERATION.STEP1.BLOCK.DATA.READ.ACTIVE
W8.02 BOOL  ; OPERATION.AUTO.CYCLE.SLAB.DATA.READ.ACTIVE
W8.03 BOOL  ; Place Holder for Incrementing (if required) Block Pointer
W8.04 BOOL  ; OPERATION.AUTO.CYCLE.SLAB.POINTER.ENABLED
W8.05 BOOL  ; OPERATION.STEP2.CALCULATE.POSITIONS
W8.06 BOOL  ; OPERATION.AUTO.CYCLE.STEP2.CALCULATE.CROSS.FORWARD.POSITION
W8.07 BOOL  ; OPERATION.AUTO.CYCLE.STEP2.CALCULATE.FIRST.CUT.POSITION
W8.08 BOOL  ; OPERATION.AUTO.CYCLE.STEP7.CALACULATE.SLAB.SIZE
W8.09 BOOL  ; OPERATION.MOVE.BLOCK.HEIGHT.TO.VERTICAL.TARGET
W8.10 BOOL  ; OPERATION.AUTO.CYCLE.SEQ.STEP5.CALULATE.CUT.HEIGHT
W8.11 BOOL  ; OPERATION.AUTO.CYCLE.CALCULATE.LONG.TARGET.PART1
W8.12 BOOL  ; OPERATION.AUTO.CYCLE.CALCULATE.FINAL.LONG.TARGET
W8.13 BOOL  ; OPERATION.AUTO.CYCLE.LAST.CUT.FOR.CURRENT.SLAB
W8.14 BOOL  ; OPERATION.AUTO.CYCLE.CURRENT.SLAB.COUNTED.EQUALS.SLAB.QTY
W8.15 BOOL  ; OPERATION.AUTO.CYCLE.INC.SLAB.PTR
W90.00 BOOL  ; Block Data Write Step 0
W90.01 BOOL  ; Slab Data Write Step 1
W90.02 BOOL  ; Change Block Offset Pointer
W90.03 BOOL  ; Read Block Data
W90.04 BOOL  ; Slab Offset Adjust
W90.05 BOOL  ; Slab Offset Pointer Update
W90.06 BOOL  ; Slab Data Read
W90.07 BOOL  ; Last Step
W9.00 BOOL  ; OPERATION.AUTO.CYCLE.DEC.SLAB.PTR
W9.01 BOOL  ; OPERATION.AUTO.CYCLE.RST.SLAB.PTR
W9.02 BOOL  ; OPERATION.AUTO.CYCLE.SLAB.PTR.CHNG
W9.03 BOOL  ; OPERATION.AUTO.CYCLE.BLOCK.POINTER.ENABLED
W9.04 BOOL  ; OPERATION.AUTO.CYCLE.INC.BLK.PTR
W9.05 BOOL  ; OPERATION.AUTO.cYCLE.DEC.BLK.PTR
W9.06 BOOL  ; OPERATION.AUTO.CYCLE.RST.BLK.PTR
W9.07 BOOL  ; OPERATION.AUTO.CYCLE.BLOCK.CHANGE
W9.08 BOOL  ; OPERATION.AUTO.CYCLE.BLOCK.COUNTED.EQUALS.BLOCK.QTY
W9.10 BOOL  ; OPERATION.AUTO.CYCLE.SEQUENCE.COMPLETE
BLADE_KERF D210 CHANNEL  ; BLADE.KERF.VALUE
BLADE_KERF_WORK_REAL D20 REAL  ; BLADE.KERF.VALUE.FLOAT.WORKING
BLK_DATA_END_ADR D1999 CHANNEL  ; Block Datat Tabe dimension end address
BLK_DATA_STRT_ADR D1000 CHANNEL  ; Dimension the Block Data Table - Start Address
BLK_DAT_RD_INIT H90.01 BOOL  ; Block Data Read Initiated
BLK_DAT_WRT_INIT H90.00 BOOL  ; Block Data Write Initiated
Block_Pointer Calculate_Pointer
CONST_MM_TO_INCH_DIV D7008 CHANNEL  ; CONST.MM.TO.INCH.DIVISOR
CUT_DEPTH D211 CHANNEL  ; CUT.DEPTH.VALUE.PROGRAMMED
CUT_DEPTH_VAL_FLT D22 REAL  ; CUT.DEPTH.VALUE.FLOAT
CUT_TRGT_CUR D212 CHANNEL  ; CUT.TARGET.CURRENT
DI_ENC_0_A 0.08 BOOL  ; _Ve
DI_ENC_0_B 0.09 BOOL  ; ENCODER.0.B
DI_ENC_0_Z 0.03 BOOL  ; ENCODER.0.Z
DI_ENC_1_A 0.06 BOOL  ; ENCODER.1.A
DI_ENC_1_B 0.07 BOOL  ; ENCODER.1.B
DI_ENC_1_Z 0.02 BOOL  ; ENCODER.1.Z
DI_FLOW_SW 1.00 BOOL  ; WATER.FLOW.SWITCH
DI_LONG_AXIS_HOME_SENS 1.01 BOOL  ; DI.LONG.AXIS.HOME.SENSOR
DI_LONG_AXIS_INDEX_CPT 0.04 BOOL  ; DI.LONG.AXIS.INDEX.COMPLETE
DI_LONG_MASTER_DRV_OK 0.10 BOOL  ; IO.LONG.AXIS.MASTER.DRIVE.OKAY.INPUT
DI_LONG_SLAVE_DRV_OK 0.01 BOOL  ; IO.LONG.SLAVE.DRIVE.OKAY.INPUT
DI_MCR_ON 0.00 BOOL  ; MCR.ON.POWER.ON
DI_SAFETY_ITLK 1.02 BOOL  ; SAFETY.GATE.INTERLOCK.INPUT
DI_SFT_STRT_FLT 0.11 BOOL  ; SAW.SOFT.START.FAULT
DI_TRANS_AXIS_DRV_OK 1.04 BOOL  ; IO.TRANSVERSE.AXIS.DRIVE.OKAY.INPUT
DI_TRANS_FWD 1.06 BOOL  ; TRANSVERSE.AXIS.FORWARD.LIMT.PROXIMITY
DI_TRANS_HOME 1.05 BOOL  ; TRANSVERSE.AXIS.HOME.PROXIMITY
DI_VERT_AXIS_DRV_OK 1.10 BOOL  ; IO.VERTICAL.AXIS.DRIVE.OKAY.INPUT
DI_VERT_FWD 1.08 BOOL  ; VERTICAL.AXIS.FORWARD.LIMIT
DI_VERT_HOME 1.07 BOOL  ; VERTICAL.AXIS.HOME.PROXIMITY
DO_ALARM_ANNUN 101.01 BOOL  ; ALARM.ANNUNCIATOR
DO_LAZER_ON 101.07 BOOL  ; LASER.ON
DO_LONG_AXIS_DRV_INDEX_CMD 101.02 BOOL  ; LONG.AXIS.MASTER.DRV.INDEX.COMMAND
DO_LONG_AXIS_HOME_INIT 101.06 BOOL  ; LONG.AXIS.MASTER.DRV.INITIATE.HOME.MOVE
DO_LONG_AXIS_JOG_LEFT 101.04 BOOL  ; LONG.AXIS.MASTER.DRV.JOG.LEFT
DO_LONG_AXIS_JOG_RIGHT 101.05 BOOL  ; LONG.AXIS.MASTER.DRV.JOG.RIGHT
DO_SFT_STRT_RUN 100.01 BOOL  ; SOFT.START.RUN
DO_SFT_STRT_STP 101.00 BOOL  ; SOFT.START.STOP
DO_TRANS_AXIS_FWD 100.04 BOOL  ; TRANSVERSE.AXIS.FORWARD
DO_TRANS_AXIS_REV 100.05 BOOL  ; TRANSVERSE.AXIS.REVERSE
DO_VERT_AXIS_BRK 101.03 BOOL  ; VERTICAL.AXIS.BRAKE.RELEASE
DO_VERT_AXIS_LWR 100.03 BOOL  ; VERTICAL.AXIS.LOWER
DO_VERT_AXIS_RAISE 100.02 BOOL  ; VERTICAL.AXIS.RAISE
DO_VERT_AXIS_SPD_SEL 100.06 BOOL  ; VERTICAL.AXIS.SPEED.SELECT.HIGH
DO_WATER_VLV 100.00 BOOL  ; WATER.VALVE
GLOBAL_HOME_REQUEST W0.15 BOOL  ; GLOBAL.HOME.REQUEST
HSC0_Init HSC0_INIT
HSC0_Init_Plx W0.00 BOOL  ; HSC0 Initialised at Power Up
HSC0_PWR_INIT H0.00 BOOL  ; HSC.0.PWR.INIT
HSC1_Init HSC1_INIT
HSC1_Init_Plx W1.00 BOOL  ; HSC1 Initialised at power up
HSC1_PWR_INIT H0.01 BOOL  ; HSC.1.PWR.INIT
IO_LAZER_PWR_OK H15.00 BOOL  ; IO.LAZER.POWER.OKAY
IO_LAZER_SG_OK H15.01 BOOL  ; IO.LAZER.SAFETY.GATE.OKAY
IO_SAW_NOT_SAFE_TO_RUN H13.03 BOOL  ; IO.SAW.NOT.SAFE.TO.RUN
IO_SAW_PWR_OK H13.00 BOOL  ; IO.SAW.POWER.OKAY
IO_SAW_SAFE_TO_RUN H13.02 BOOL  ; IO.SAW.SAFE.TO.RUN
IO_SAW_SG_OK H13.01 BOOL  ; IO.SAW.SAFETY.GATE.OKAY
IO_Saw_Safe_To_Run Op_2_State
IO_WTR_PWR_OK H14.00 BOOL  ; IO.WATER.POWER.OKAY
IO_WTR_SG_OK H14.01 BOOL  ; IO.WATER.SAFETY.GATE.OKAY
LAXISMFDBK A276 CHANNEL  ; LONG.AXIS.MASTER.FEEDBACK
MAIN_PWR_ERR W0.05 BOOL  ; MAIN.POWER.ERR
MC_AXIS_DRV_STP_STATE H11.12 BOOL  ; MC.VERTICAL.AXIS.DRIVE.STOP.STATE
MC_AXIS_LONG_FDBK D5000 WORD  ; MC.LONG.AXIS.FEEDBACK
MC_LONG_AXIS_AUTO_NOK H10.03 BOOL  ; MC.LONG.AXIS.AUTO.NOT.OKAY
MC_LONG_AXIS_AUTO_OK H10.02 BOOL  ; MC.LONG.AXIS.AUTO.OKAY
MC_LONG_AXIS_DRV_ACT 302.00 BOOL  ; MC.LONG.AXIS.DRIVE.ACTIVE
MC_LONG_AXIS_DRV_AT_ZERO 303.00 BOOL  ; MC.LONG.AXIS.DRIVE.AT.ZERO.SPEED
MC_LONG_AXIS_DRV_EN 304.00 BOOL  ; MC.LONG.AXIS.DRV.ENABLE
MC_LONG_AXIS_DRV_ERR H10.05 BOOL  ; MC.LONG.AXIS.DRIVE.ERROR
MC_LONG_AXIS_DRV_JOG_PLUS_INPUT_MON 324.00 BOOL  ; MC.LONG.AXIS.DRIVE.JOG.PLUS.INPUT.STATE.MONITOR
MC_LONG_AXIS_DRV_MAINS_LOSS 315.00 BOOL  ; MC.LONG.AXIS.MAINS.LOSS.FAULT
MC_LONG_AXIS_DRV_OK 301.00 BOOL  ; MC.LONG.AXIS.DRIVE.OKAY
MC_LONG_AXIS_DRV_OKAY H10.04 BOOL  ; MC.LONG.AXIS.DRIVE.OKAY
MC_LONG_AXIS_DRV_OL 317.00 BOOL  ; MC.LONG.AXIS.DRIVE.OVERLOAD.FAULT
MC_LONG_AXIS_DRV_RST 333.00 BOOL  ; MC.LONG.AXIS.DRIVE.RESET
MC_LONG_AXIS_DRV_RST_EN H10.11 BOOL  ; MC.LONG.AXIS.DRIVE.RESET.ENABLED
MC_LONG_AXIS_DRV_STOP_NOT 310.00 BOOL  ; MC.LONG.AXIS.DRIVE.STOP.NOT
MC_LONG_AXIS_DRV_UV 316.00 BOOL  ; MC.LONG.AXIS.DRIVE.BUS.UNDER.VOLTAGE.ERROR
MC_LONG_AXIS_DRV_WRN 319.00 BOOL  ; MC.LONG.AXIS.DRIVE.WARNING.[FAULT EXISTS]
MC_LONG_AXIS_ERR H10.14 BOOL  ; LONG.AXIS.ERROR.EXISTS
MC_LONG_AXIS_EZMTN_ERR 314 INT  ; MC.LONG.AXIS.DRIVE.EZMOTION.MODULE.ERROR
MC_LONG_AXIS_EZMTN_STATUS 312 LINT  ; MC.LONG.AXIS.DRIVE.EZMOTION.MODULE.STATUS
MC_LONG_AXIS_FDBK_REAL D5006 REAL  ; MC.LONG.AXIS.FEEDBACK.REAL
MC_LONG_AXIS_FDBK_REAL_SCALED D5010 REAL  ; MC.LONG.AXIS.FEEDBACK.SCALED
MC_LONG_AXIS_GATE_OK H10.01 BOOL  ; LONG.AXIS.SAFETY.GATE.OKAY
MC_LONG_AXIS_HOME_ACT H20.01 BOOL  ; MC.LONG.AXIS.HOMING.ACTIVE
MC_LONG_AXIS_HOME_CMD_INT H10.08 BOOL  ; MC.LONG.AXIS.HOME.COMMAND.INTERNAL
MC_LONG_AXIS_HOME_CMPLT H20.02 BOOL  ; MC.LONG.AXIS.HOMING.COMPLETED
MC_LONG_AXIS_HOME_EN H10.12 BOOL  ; MC.LONG.AXIS.HOME.INSTRUCTION.ENABLED
MC_LONG_AXIS_HOME_ERR H20.03 BOOL  ; MC.LONG.AXIS.HOMING.ERROR.OCCURED
MC_LONG_AXIS_HOME_INIT_MON 325.00 BOOL  ; MC.LONG.AXIS.HOME.INITIATE.INPUT.MONITOR
MC_LONG_AXIS_HOME_INIT_REQ H20.00 BOOL  ; MC.LONG.AXIS.HOME.INITIALISE.REQUEST
MC_LONG_AXIS_HOME_SENSOR_MON 326.00 BOOL  ; MC.LONG.AXIS.DRIVE.HOME.SENSOR.INPUT.MONITOR
MC_LONG_AXIS_JOGR_CMD H10.07 BOOL  ; MC.LONG.AXIS.JOG.RIGHT.COMMAND
MC_LONG_AXIS_JOG_ACT H10.09 BOOL  ; MC.LONG.AXIS.JOG.ACTIVE
MC_LONG_AXIS_JOG_EN H10.06 BOOL  ; MC.LONG.AXIS.JOG.ENABLED
MC_LONG_AXIS_JOG_ERR H10.10 BOOL  ; MC.LONG.AXIS.JOG.ERROR
MC_LONG_AXIS_JOG_MIN_INPUT_MON 323.00 BOOL  ; MC.LONG.AXIS.DRV.JOG.MINUS.INPUT.MONITOR
MC_LONG_AXIS_MIN_LIM_MON 321.00 BOOL  ; MC.LONG.AXIS.DRIVE.MINUS.LIMIT.ACTIVE.MONITOR
MC_LONG_AXIS_MODID 311 INT  ; MC.LONG.AXIS.DRIVE.EZMOTION.MODULE.ID
MC_LONG_AXIS_PGM_INIT_MON 320.00 BOOL  ; MC.LONG.AXIS.DRIVE.EZMOTION.PROGRAM.INITIATE.MONITOR
MC_LONG_AXIS_PLUS_LIM_MON 322.00 BOOL  ; MC.LONG.AXIS.PLUS.LIMIT.ACTIVE.MONITOR
MC_LONG_AXIS_POS_REF_CMD D4 WORD  ; MC.LONG.AXIS.POSITION.REFERENCE.COMMAND.VALUE
MC_LONG_AXIS_PWR_OK H10.00 BOOL  ; LONG.AXIS.POWER.OKAY
MC_LONG_AXIS_RDY H10.15 BOOL  ; LONG.AXIS.MOTION.READY
MC_LONG_AXIS_RESET_CMD MC_Axis_Reset
MC_LONG_AXIS_TEMP_FLT 318.00 BOOL  ; MC.LONG.AXIS.DRIVE.OVER.TEMPERATURE.FAULT
MC_Long_Axis_Drv_OK Op_2_State
MC_Long_Axis_Home_Func MC_Axis_Srv_Home
MC_Op_Long_Axis_Jog MC_Axis_Jog
MC_Op_Trans_Axis_Jog_Cmd MC_Axis_Jog
MC_Op_Vert_Axis_Jog_Cmd MC_Axis_Jog
MC_PERM_TRANS_AXIS_AUTO_NOK H12.03 BOOL  ; MC.PERMISSIVE.TRANSVERSE.AXIS.AUTO.NOK
MC_PERM_TRANS_AXIS_AUTO_OK H12.02 BOOL  ; MC.PERMISSIVE.TRANSVERSE.AXIS.AUTO.OK
MC_TRANS_AXIS_DRV_ACT 402.00 BOOL  ; MC.TRANSVERSE.AXIS.DRIVE.ACTIVE
MC_TRANS_AXIS_DRV_AT_ZERO_SPD 403.00 BOOL  ; MC.TRANSVERSE.AXIS.DRIVE.AT.ZERO.SPEED
MC_TRANS_AXIS_DRV_ERR H12.05 BOOL  ; MC.TRANSVERSE.AXIS.DRIVE.ERROR
MC_TRANS_AXIS_DRV_GNRL_ERR 419.00 BOOL  ; MC.TRANSVERSE.AXIS.DRIVE.GENERAL.ERROR
MC_TRANS_AXIS_DRV_MAINS_LOSS 415.00 BOOL  ; MC.TRANSVERSE.AXIS.DRIVE.MAINS.LOSS
MC_TRANS_AXIS_DRV_NOT_STOP 410.00 BOOL  ; MC.TRANSVERSE.AXIS.DRIVE.NOT.STOP
MC_TRANS_AXIS_DRV_OK 401.00 BOOL  ; MC.TRANSVERSE.AXIS.DRIVE.OKAY.STATUS
MC_TRANS_AXIS_DRV_OK_PERM H12.04 BOOL  ; MC.PERMISSIVE.TRANSVERSE.AXIS.DRIVE.OKAY
MC_TRANS_AXIS_DRV_OL 417.00 BOOL  ; MC.TRANSVERSE.AXIS.DRIVE.OVERLOAD.ERROR
MC_TRANS_AXIS_DRV_PREC_REF_SEL 444.00 BOOL  ; MC.TRANSVERSE.AXIS.DRIVE.PRECISION.REFERENCE.SELECT
MC_TRANS_AXIS_DRV_RESET 433.00 BOOL  ; MC.TRANSVERSE.AXIS.DRIVE.ERROR.RESET
MC_TRANS_AXIS_DRV_RST MC_Axis_Reset
MC_TRANS_AXIS_DRV_RUN_FWD 405.00 BOOL  ; MC.TRANSVERSE.AXIS.DRIVE.RUN.FORWARD
MC_TRANS_AXIS_DRV_RUN_REV 407.00 BOOL  ; MC.TRANSVERSE.AXIS.DRIVE.RUN.REVERSE
MC_TRANS_AXIS_DRV_STP_STATE H12.12 BOOL  ; MC.TRANSVERSE.AXiS.DRIVE.STOP.STATE
MC_TRANS_AXIS_DRV_TEMP_ERR 418.00 BOOL  ; MC.TRANSVERSE.AXIS.DRIVE.TEMPERATURE.ERROR
MC_TRANS_AXIS_ERR H12.14 BOOL  ; TRANSVERSE.AXIS.ERROR.EXISTS
MC_TRANS_AXIS_FDBK_INTRM2 D28 LINT  ; MC.TRANSVERSE.AXIS.VELOCITY.FEEDBACK.INTERIM2
MC_TRANS_AXIS_FT_P_MIN D30 INT  ; MC.TRANSVERSE.AXIS.FEET.PER.MIN
MC_TRANS_AXIS_HOME_ACT H22.01 BOOL  ; MC.TRANSVERSE.AXIS.HOMING.ACTIVE
MC_TRANS_AXIS_HOME_CMP H22.02 BOOL  ; MC.TRANSVERSE.AXIS.HOMING.COMPLETED
MC_TRANS_AXIS_HOME_ERR H22.03 BOOL  ; MC.TRANSVERSE.AXIS.HOMING.ERROR
MC_TRANS_AXIS_HOME_INIT_REQ H22.00 BOOL  ; MC.TRANSVERSE.AXIS.HOME.INITIALISE.REQUEST
MC_TRANS_AXIS_JOG_ACT H12.09 BOOL  ; MC.TRANSVERSE.AXIS.JOG.COMMAND.ACTIVE
MC_TRANS_AXIS_JOG_CMD_ERR H12.10 BOOL  ; MC.TRANSVERSE.AXIS.JOG.COMMAND.ERROR
MC_TRANS_AXIS_JOG_EN H12.06 BOOL  ; MC.TRANSVERSE.AXIS.JOG.ENABLED
MC_TRANS_AXIS_JOG_FWD 406.00 BOOL  ; MC.TRANSVERSE.AXIS.DRIVE.JOG.FORWARD
MC_TRANS_AXIS_JOG_REV 408.00 BOOL  ; MC.TRANSVERSE.AXIS.DRIVE.JOG.REVERSE
MC_TRANS_AXIS_NOT_STP_MON H12.11 BOOL  ; MC.TRANSVERSE.AXIS.DRIVE.NOT.STOP.MONITOR
MC_TRANS_AXIS_PWR_OK H12.00 BOOL  ; TRANSVERSE.AXIS.POWER.OKAY
MC_TRANS_AXIS_READY H12.15 BOOL  ; MC.TRANSVERSE.READY
MC_TRANS_AXIS_SAFETY_GATE_OK H12.01 BOOL  ; TRANSVERSE.AXIS.SAFETY.GATE.OKAY
MC_TRANS_AXIS_VEL_FDBK_INTRM D26 LINT  ; MC.TRANSVERSE.AXIS.VELOCITY.FEEDBACK.INTERIM
MC_TRANS_POS_FDBK_SCALED D6010 REAL  ; MC.TRANSVERSE.AXIS.POSITION.FEEDBACK.INCHES.SCALED.REAL
MC_TRAN_AXIS_DRV_EN 404.00 BOOL  ; MC.TRANSVERSE.AXIS.DRIVE.ENABLE
MC_VERT_AXISDRV_NOT_STP 510.00 BOOL  ; MC.VERTICAL.AXIS.DRIVE.NOT.STOP
MC_VERT_AXIS_AUTO_OK H11.02 BOOL  ; MC.VERTICAL.AXIS.AUTO.OK
MC_VERT_AXIS_DRV_ACT 502.00 BOOL  ; MC.VERTICAL.AXIS.DRIVE.ACTIVE
MC_VERT_AXIS_DRV_AT_ZERO_SPD 503.00 BOOL  ; MC.VERTICAL.AXIS.DRIVE.AT.ZERO.SPEED
MC_VERT_AXIS_DRV_EN 504.00 BOOL  ; MC.VERTICAL.AXIS.DRIVE.ENABLE
MC_VERT_AXIS_DRV_ERR H11.05 BOOL  ; MC.VERTICAL.AXIS.DRIVE.ERROR
MC_VERT_AXIS_DRV_GNRL_ERR 519.00 BOOL  ; MC.VERTICAL.AXIS.DRIVE.GENERAL.ERROR
MC_VERT_AXIS_DRV_MAINS_LOSS 515.00 BOOL  ; MC.VERTICAL.AXIS.DRIVE.MAINS.LOSS
MC_VERT_AXIS_DRV_NOT_STP_MON H11.11 BOOL  ; MC.VERT.AXIS.DRV.NOT.STP.MON
MC_VERT_AXIS_DRV_OK 501.00 BOOL  ; MC.VERTICAL.AXIS.DRIVE.OKAY
MC_VERT_AXIS_DRV_OK_PERM H11.04 BOOL  ; MC.VERTICAL.AXIS.DRIVE.OKAY.PERMISSIVE
MC_VERT_AXIS_DRV_OL 517.00 BOOL  ; MC.VERTICAL.AXIS.DRIVE.OVERLOAD.ERROR
MC_VERT_AXIS_DRV_PREC_REF_SEL 544.00 BOOL  ; MC.VERTICAL.AXIS.DRIVE.PRECISION.REFERENCE.SELECT
MC_VERT_AXIS_DRV_RESET 533.00 BOOL  ; MC.VERTICAL.AXIS.DRIVE.RESET
MC_VERT_AXIS_DRV_RUN_REV 507.00 BOOL  ; MC.VERTICAL.AXIS.DRIVE.RUN.REVERSE
MC_VERT_AXIS_DRV_TEMP_ERR 518.00 BOOL  ; MC.VERTICAL.AXIS.DRIVE.TEMPERATURE.ERROR
MC_VERT_AXIS_ERR H11.14 BOOL  ; MC.VERTICAL.AXIS.ERROR
MC_VERT_AXIS_FDBK_BALLSC_REV_REAL D7004 CHANNEL  ; MC.VERTICAL.POSITION.FEEDBACK.BALLSCREW.REVOLUTIONS.REAL
MC_VERT_AXIS_FDBK_REAL_SCALED D7010 REAL  ; MC.VERTICAL.AXIS.FEEDBACK.REAL.SCALED.INCH
MC_VERT_AXIS_HOME_ACT H21.01 BOOL  ; MC.VERTICAL.AXIS.HOMING.ACTIVE
MC_VERT_AXIS_HOME_CMP H21.02 BOOL  ; MC.VERTICAL.AXIS.HOMING.COMPLETED
MC_VERT_AXIS_HOME_ERR H21.03 BOOL  ; MC.VERTICAL.AXIS.HOMING.ERROR
MC_VERT_AXIS_HOME_INIT_REQ H21.00 BOOL  ; MC.VERTICAL.AXIS.HOME.INITIALISE.REQUEST
MC_VERT_AXIS_JOG_ACT H11.09 BOOL  ; MC.VERTICAL.AXIS.JOG.ACTIVE
MC_VERT_AXIS_JOG_EN H11.06 BOOL  ; MC.VERTICAL.AXIS.JOG.ENABLED
MC_VERT_AXIS_JOG_FWD 506.00 BOOL  ; MC.VERTICAL.AXIS.DRIVE.JOG.FORWARD
MC_VERT_AXIS_JOG_REV 508.00 BOOL  ; MC.VERTICAL.AXIS.JOG.REVERSE
MC_VERT_AXIS_JO_CMD_ERR H11.10 BOOL  ; MC.VERTICAL.AXIS.JOG.COMMAND.ERROR
MC_VERT_AXIS_POS_ACT_SCALED_MM D7006 CHANNEL  ; MC.VERTICAL.POSITION.ACTUAL.SCALED.MM
MC_VERT_AXIS_POS_FDBK_GB_SCALED_REAL D7002 CHANNEL  ; MC.VERTICAL.AXIS.POSITION.REVOLUTION.REAL
MC_VERT_AXIS_POS_FDBK_RAW D7000 CHANNEL  ; MC.VERTICAL.AXIS.POSITION.FEEDBACK.RAW.REAL
MC_VERT_AXIS_PWR_OK H11.00 BOOL  ; VERTICAL.AXIS.POWER.OKAY
MC_VERT_AXIS_RDY H11.15 BOOL  ; MC.VERTICAL.AXIS.READY
MC_VERT_AXIS_RST MC_Axis_Reset
MC_VERT_AXIS_RUN_FWD 505.00 BOOL  ; MC.VERTICAL.AXIS.DRIVE.RUN.FORWARD
MC_VERT_AXIS_SAFETY_GATE_OK H11.01 BOOL  ; VERTICAL.AXIS.SAFETY.GATE.OKAY
MODE_AUTO_IND W130.14 BOOL  ; AUTOMATIC.MODE.INDICATOR
MODE_MAN_IND W130.13 BOOL  ; MANUAL.MODE.INDICATOR
MODE_SEL_AUTO W0.09 BOOL  ; MODE.SELECT.AUTOMATIC
MODE_SEL_AUTO_EN W0.11 BOOL  ; MODE.SELECT.AUTO.MODE.ENABLED
MODE_SEL_EN W0.07 BOOL  ; MODE.SELECT.ENABLED
MODE_SEL_MAN W0.08 BOOL  ; MODE.SELECT.MANUAL
MODE_SEL_MAN_EN W0.10 BOOL  ; MODE.SELECT.MANUAL.MODE.ENABLED
Message_Display Op_Message
Mode_Select Op_Mode_Sel
OI_ALARM_MESSAGE_SELECT Op_Message
OI_ALM_CLR W111 WORD  ; OI.ALARM.MESSAGE.COLOUR
OI_ALM_IND W130.15 BOOL  ; OI.ALARM.INDICATOR.ACTIVE
OI_ALM_SEL W110 WORD  ; OI.ALARM.MESSAGE.SELECT
OI_CTL_ALM_RESET W121.08 BOOL  ; OPERATION.CONTROL.ALARM.RESET.PB
OI_CTL_TRANS_AXIS_HOME_PB W120.12 BOOL  ; OI.TRANSVERSE.AXIS.HOME.PB
OI_CTL_WORD_1 W120 WORD  ; OI.CONTROL.WORD.1
OI_CTL_WORD_2 W121 WORD  ; OI.CONTROL.WORD.2
OI_CTRL_CYCLE_START W120.02 BOOL  ; OI.CONTROL.AUTOMATIC.CYCLE.START.PB
OI_CTRL_CYCLE_STOP_PB W120.01 BOOL  ; OI.CONTROL.AUTOMATIC.CYCLE.STOP.PB
OI_CTRL_H_A_SEL W120.00 BOOL  ; OI.CONTROL.HAND.AUTO.SELECTOR
OI_CTRL_MAC_STOP W120.03 BOOL  ; OI.CONTROL.AUTOMATIC.CYCLE.MACHINE.STOP
OI_HOME_ALL_PB W120.04 BOOL  ; OI.HOME.ALL.PB
OI_IND_WORD_1 W130 WORD  ; OI.INDICATE.WORD.1
OI_IND_WORD_2 W131 WORD  ; OI.INDICATE.WORD.2
OI_LONG_AXIS_HOME_REQ W121.01 BOOL  ; OI.LING.AXIS.HOME.REQUEST.PB
OI_LONG_AXIS_JOG_MINUS W120.15 BOOL  ; OI.LONG.AXIS.JOG.MINUS.PB
OI_LONG_AXIS_JOG_PLUS W121.00 BOOL  ; OI.LONG.AXIS.JOG.PLUS.PB
OI_MSG_CLR W101 INT  ; OI.MESSAGE.COLOUR
OI_MSG_SEL W100 INT  ; OI.MESSAGE.SELECT
OI_SAW_CUR_ACT_SCL D140 LWORD  ; OI.SAW.CURRENT.SCALED
OI_SAW_CUR_CALC D120 LWORD  ; OI.SCALING.SAW.CURRENT.PART1
OI_SAW_STP_PB W120.08 BOOL  ; OI.SAW.STOP.PB
OI_SAW_STRT_PB W120.07 BOOL  ; OI.SAW.START.PB
OI_SET_FIRST_CUT W121.06 BOOL  ; OI.SET.FIRST.CUT.REQUEST
OI_Saw_Mach_Stop Op_2_State
OI_TRANS_AXIS_JOG_HOME_PB W120.13 BOOL  ; OI.TRANSVERSE.AXIS.JOG.HOME.PB
OI_TRANS_AXIS_JO_FWD_PB W120.14 BOOL  ; OI.TRANSVERSE.AXIS.JOG.FORWARD.PB
OI_VERT_AXIS_JOG_FWD_PB W120.11 BOOL  ; OI.VERTICAL.AXIS.JOG.FORWARD.PB
OI_VERT_AXIS_JOG_HOME_PB W120.10 BOOL  ; OI.VERTICAL.AXIS.JOG.HOME.PB
OI_WTR_ON_SEL W120.06 BOOL  ; OI.WATER.ON.SELECTOR
OOI_LAZER_ON_SEL W120.05 BOOL  ; OI.LAZER.ON.SELECTOR
OPERATION_AUTO_CYC_INCREMENT_BLOCK Calculate_Pointer
OPERATION_AUTO_CYC_INCREMENT_SLAB Calculate_Pointer
OP_ALARM_RESET H0.13 BOOL  ; OPERATION.ALARM.RESET.REQUEST
OP_ALARM_STATE_ACTIVE H0.15 BOOL  ; OP.ALARM.STATE.ACTIVE(FAULTED)
OP_ALMS_RES_EN Op_2_State
OP_ALM_MON_EN H0.12 BOOL  ; OP.ALARM.MONITORING.ENABLED
OP_ALRM_MON_ACT H0.14 BOOL  ; OPERATION.ALARM.CONDITION.MONITRING.ACTIVE
OP_AUTO_BLK_ID D4114 INT  ; OPERATION.AUTO.CYCLE.BLOCK.ID
OP_AUTO_CYC_BLK_CNT D4102 INT  ; OPERATION.AUTO.CYCLE.BLOCK.COUNT
OP_AUTO_CYC_BLK_FCUT D4106 INT  ; OPERATION.AUTO.CYCLE.BLOCK.FIRST.CUT.WORKING
OP_AUTO_CYC_BLK_HEIGHT D4100 INT  ; OPERATION.AUTO.CYCLE.BLOCK.HEIGHT.WORKING
OP_AUTO_CYC_BLK_LEN D4104 INT  ; OPERATION.AUTO.CYCLE.BLOCK.TRANSVERSE.AXIS.STOP.POSITION.WORKING
OP_AUTO_CYC_BLK_QTY D4116 INT  ; OPERATION.AUTO.CYCLE.BLOCK.QUANTITY
OP_AUTO_CYC_BLK_SLABQ D4108 INT  ; OPERATION.AUTO.CYCLE.CURRENT.BLOCK.SLAB.QUANTITY
OP_AUTO_CYC_SLAB_ID D4118 INT  ; OPERATION.AUTO.CYCLE.SLAB.ID
OP_AUTO_CYC_SLAB_QTY D4112 INT  ; OPERATION.AUTO.CYCLE.CURRENT.SLABS.QUANTITY
OP_AUTO_CYC_SLAB_SZ D4110 INT  ; OPERATION.AUTO.CYCLE.CURRENT.SLAB.SIZE
OP_Alarm_Monitor Op_Alarm_Monitor
OP_CTL_AUTO_CYCLE_RUN_STEP1 W6.03 BOOL  ; OP.CONTROL.AUTO.CYCLE.RUN.EXECUTE.STEP1
OP_CTL_AUTO_CYC_STRTUP_STATE W6.00 BOOL  ; OP.CONTROL.AUTO.CYCLE.START.STATE
OP_CTL_AUTO_CYC_STRT_SAW_RUN W6.01 BOOL  ; OP.CONTROL.AUTO.CYCLE.SAW.START.STEP.DONE
OP_CTL_AUTO_CYC_STRT_WATER_ON W6.02 BOOL  ; OP.CONTROL.AUTO.CYCLE.START.WATER.COMPLETE
OP_CTRL_LONG_AXIS_TARG_REAL D5100 REAL  ; OPERATION.CONTROL.LONG.AXIS.TARGET.REAL
OP_CYCLE_RUN Op_Cyc_Run
OP_CYCLE_START Op_Cyc_Strt
OP_CYC_STOP Op_Cyc_Stp
OP_FIRST_CYC_CMPLT H0.02 BOOL  ; FIRST.CYCLE.COMPLETED
OP_Mode_Indicator Op_Mode_Ind
OP_PGM_CHK_SLAB10_EN H25.09 BOOL  ; OPERATION.ENABLE.SLAB10.DISPLAY
OP_PGM_CHK_SLAB11_EN H25.10 BOOL  ; OPERATION.ENABLE.SLAB11.DISPLAY
OP_PGM_CHK_SLAB12_EN H25.11 BOOL  ; OPERATION.ENABLE.SLAB12.DISPLAY
OP_PGM_CHK_SLAB13_EN H25.12 BOOL  ; OPERATION.ENABLE.SLAB13.DISPLAY
OP_PGM_CHK_SLAB14_EN H25.13 BOOL  ; OPERATION.ENABLE.SLAB14.DISPLAY
OP_PGM_CHK_SLAB15_EN H25.14 BOOL  ; OPERATION.ENABLE.SLAB15.DISPLAY
OP_PGM_CHK_SLAB16_EN H25.15 BOOL  ; OPERATION.ENABLE.SLAB16.DISPLAY
OP_PGM_CHK_SLAB17_EN H26.00 BOOL  ; OPERATION.ENABLE.SLAB17.DISPLAY
OP_PGM_CHK_SLAB18_EN H26.01 BOOL  ; OPERATION.ENABLE.SLAB18.DISPLAY
OP_PGM_CHK_SLAB19_EN H26.02 BOOL  ; OPERATION.ENABLE.SLAB19.DISPLAY
OP_PGM_CHK_SLAB1_EN H25.00 BOOL  ; OPERATION.ENABLE.SLAB1.DISPLAY
OP_PGM_CHK_SLAB20_EN H26.03 BOOL  ; OPERATION.ENABLE.SLAB20.DISPLAY
OP_PGM_CHK_SLAB21_EN H26.04 BOOL  ; OPERATION.ENABLE.SLAB21.DISPLAY
OP_PGM_CHK_SLAB22_EN H26.05 BOOL  ; OPERATION.ENABLE.SLAB22.DISPLAY
OP_PGM_CHK_SLAB23_EN H26.06 BOOL  ; OPERATION.ENBLE.SLAB23.DISPLAY
OP_PGM_CHK_SLAB24_EN H26.07 BOOL  ; OPERATION.ENABLE.SLAB24.DISPLAY
OP_PGM_CHK_SLAB25_EN H26.08 BOOL  ; OPERATION.ENABLE.SLAB25.DISPLAY
OP_PGM_CHK_SLAB26_EN H26.09 BOOL  ; OPERATION.ENABLE.SLAB26.DISPLAY
OP_PGM_CHK_SLAB27_EN H26.10 BOOL  ; OPERATION.ENABLE.SLAB27.DISPLAY
OP_PGM_CHK_SLAB28_EN H26.11 BOOL  ; OPERATION.ENABLE.SLAB28.DISPLAY
OP_PGM_CHK_SLAB29_EN H26.12 BOOL  ; OPERATION.ENABLE.SLAB29.DISPLAY
OP_PGM_CHK_SLAB2_EN H25.01 BOOL  ; OPERATION.ENABLE.SLAB2.DISPLAY
OP_PGM_CHK_SLAB30_EN H26.13 BOOL  ; OPERATIOn.ENABLE.SLAB30.DISPLAY
OP_PGM_CHK_SLAB31_EN H26.14 BOOL
OP_PGM_CHK_SLAB32_EN H26.15 BOOL
OP_PGM_CHK_SLAB33_EN H27.00 BOOL
OP_PGM_CHK_SLAB34_EN H27.01 BOOL
OP_PGM_CHK_SLAB35_EN H27.02 BOOL
OP_PGM_CHK_SLAB36_EN H27.03 BOOL
OP_PGM_CHK_SLAB37_EN H27.04 BOOL
OP_PGM_CHK_SLAB39_EN H27.06 BOOL
OP_PGM_CHK_SLAB3_EN H25.02 BOOL  ; OPERATION.ENABLE.SLAB3.DISPLAY
OP_PGM_CHK_SLAB40_EN H27.07 BOOL
OP_PGM_CHK_SLAB41_EN H27.08 BOOL
OP_PGM_CHK_SLAB42_EN H27.09 BOOL
OP_PGM_CHK_SLAB43_EN H27.10 BOOL
OP_PGM_CHK_SLAB44_EN H27.11 BOOL
OP_PGM_CHK_SLAB45_EN H27.12 BOOL
OP_PGM_CHK_SLAB46_EN H27.13 BOOL
OP_PGM_CHK_SLAB47_EN H27.14 BOOL
OP_PGM_CHK_SLAB48_EN H27.15 BOOL
OP_PGM_CHK_SLAB49_EN H28.00 BOOL
OP_PGM_CHK_SLAB4_EN H25.03 BOOL  ; OPERATION.ENABLE.SLAB4.DISPLAY
OP_PGM_CHK_SLAB50_EN H28.01 BOOL
OP_PGM_CHK_SLAB51_EN H28.02 BOOL
OP_PGM_CHK_SLAB52_EN H28.03 BOOL
OP_PGM_CHK_SLAB53_EN H28.04 BOOL
OP_PGM_CHK_SLAB54_EN H28.05 BOOL
OP_PGM_CHK_SLAB55_EN H28.06 BOOL
OP_PGM_CHK_SLAB56_EN H28.07 BOOL
OP_PGM_CHK_SLAB57_EN H28.08 BOOL
OP_PGM_CHK_SLAB58_EN H28.09 BOOL
OP_PGM_CHK_SLAB59_EN H28.10 BOOL
OP_PGM_CHK_SLAB5_EN H25.04 BOOL  ; OPERATION.ENABLE.SLAB5.DISPLAY
OP_PGM_CHK_SLAB60_EN H28.11 BOOL
OP_PGM_CHK_SLAB61_EN H28.12 BOOL
OP_PGM_CHK_SLAB62_EN H28.13 BOOL
OP_PGM_CHK_SLAB63_EN H28.14 BOOL
OP_PGM_CHK_SLAB64_EN H28.15 BOOL
OP_PGM_CHK_SLAB65_EN H29.00 BOOL
OP_PGM_CHK_SLAB66_EN H29.01 BOOL
OP_PGM_CHK_SLAB67_EN H29.02 BOOL
OP_PGM_CHK_SLAB68_EN H29.03 BOOL
OP_PGM_CHK_SLAB69_EN H29.04 BOOL
OP_PGM_CHK_SLAB6_EN H25.05 BOOL  ; OPERATION.ENABLE.SLAB6.DISPLAY
OP_PGM_CHK_SLAB70_EN H29.05 BOOL
OP_PGM_CHK_SLAB71_EN H29.06 BOOL
OP_PGM_CHK_SLAB72_EN H29.07 BOOL
OP_PGM_CHK_SLAB73_EN H29.08 BOOL
OP_PGM_CHK_SLAB74_EN H29.09 BOOL
OP_PGM_CHK_SLAB75_EN H29.10 BOOL
OP_PGM_CHK_SLAB76_EN H29.11 BOOL
OP_PGM_CHK_SLAB77_EN H29.12 BOOL
OP_PGM_CHK_SLAB78_EN H29.13 BOOL
OP_PGM_CHK_SLAB79_EN H29.14 BOOL
OP_PGM_CHK_SLAB7_EN H25.06 BOOL  ; OPERATION.ENABLE.SLAB7.DISPLAY
OP_PGM_CHK_SLAB80_EN H29.15 BOOL
OP_PGM_CHK_SLAB81_EN H30.00 BOOL
OP_PGM_CHK_SLAB82_EN H30.01 BOOL
OP_PGM_CHK_SLAB83_EN H30.02 BOOL
OP_PGM_CHK_SLAB8_EN H25.07 BOOL  ; OPERATION.ENABLE.SLAB8.DISPLAY
OP_PGM_CHK_SLAB9_EN H25.08 BOOL  ; OERATION.ENABLE.SLAB9.DISPLAY
OP_PGM_CHK_SLAB_38_EN H27.05 BOOL
OP_Power_On_Check Op_2_State
Op_Gate_Monitor Op_2_State
Op_Long_Axis_Mach_Stop Op_2_State
Op_Mach_Stop_Water Op_2_State
Op_Perm_Long_Auto Op_2_State
Op_Trans_Auto_Ok Op_2_State
Op_Trans_Axis_Drv_Ok Op_2_State
Op_Trans_Axis_Mach_Stop Op_2_State
Op_Vert_Auto_Ok Op_2_State
Op_Vert_Axis_Mach_Stop Op_2_State
Op_Vert_Axis_Ok Op_2_State
POWER_ON W0.03 BOOL  ; POWER.ON.MAIN
SAFETY_GATE_ERR W0.06 BOOL  ; SAFETY.GATE.ERR
SAFETY_GATE_OK W0.04 BOOL  ; SAFETY.GATE.OKAY
SLAB_DATA_END_ADR D2999 CHANNEL  ; DIMENSION.SLAB.DATA.TABLE.END.ADDRESS
SLAB_DATA_START_ADR D2000 CHANNEL  ; DIMENSION.SLAB.DATA.TABLE.START.ADDRESS
Slab_Pointer Calculate_Pointer
TARGET_CURRENT_WKNG D24 REAL  ; TARGET.CURRENT.WORKING.FLOAT
TRANS_POS_FDBK A272 CHANNEL  ; TRANSVERSE.POSITION.FEEDBACK.RAW
VERT_POS_FDBK A270 CHANNEL  ; VERTICAL.POSITION.FEEDBACK.RAW

## Program Main (cyclic task 0)
; Main saw program file

### Section Init_HSC

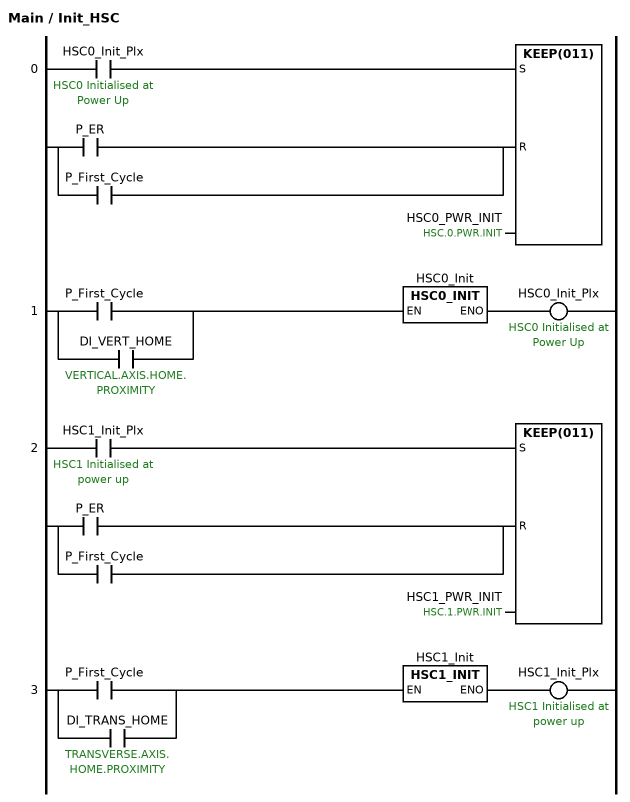
; rung 0
LD HSC0_Init_Plx  ; HSC0 Initialised at Power Up
LD P_ER
OR P_First_Cycle
KEEP(011) HSC0_PWR_INIT  ; HSC.0.PWR.INIT
; rung 1
LD P_First_Cycle
OR DI_VERT_HOME  ; VERTICAL.AXIS.HOME.PROXIMITY
CALL HSC0_Init : HSC0_INIT ()
OUT HSC0_Init_Plx  ; HSC0 Initialised at Power Up
; rung 2
LD HSC1_Init_Plx  ; HSC1 Initialised at power up
LD P_ER
OR P_First_Cycle
KEEP(011) HSC1_PWR_INIT  ; HSC.1.PWR.INIT
; rung 3
LD P_First_Cycle
OR DI_TRANS_HOME  ; TRANSVERSE.AXIS.HOME.PROXIMITY
CALL HSC1_Init : HSC1_INIT ()
OUT HSC1_Init_Plx  ; HSC1 Initialised at power up

### Section Interlock_Alarm

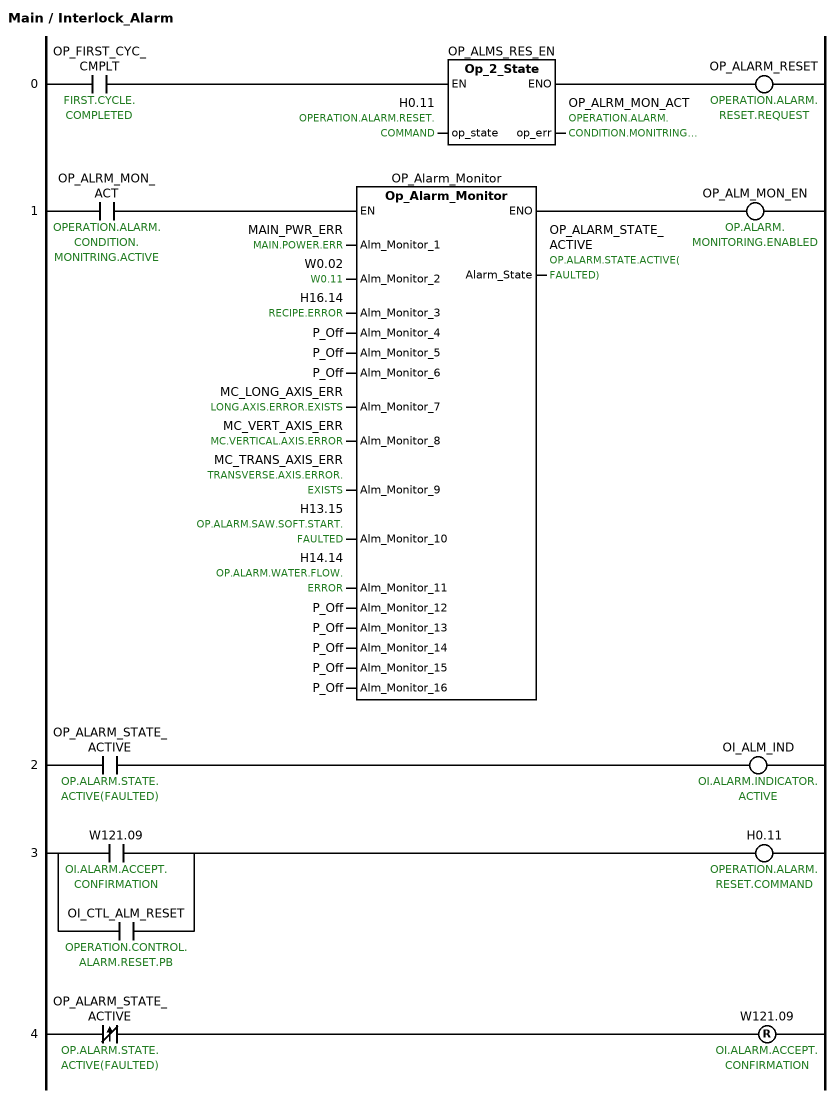
; rung 0
LD OP_FIRST_CYC_CMPLT  ; FIRST.CYCLE.COMPLETED
CALL OP_ALMS_RES_EN : Op_2_State (op_state := H0.11, op_err => OP_ALRM_MON_ACT)  ; OPERATION.ALARM.RESET.COMMAND, OPERATION.ALARM.CONDITION.MONITRING.ACTIVE
OUT OP_ALARM_RESET  ; OPERATION.ALARM.RESET.REQUEST
; rung 1
LD OP_ALRM_MON_ACT  ; OPERATION.ALARM.CONDITION.MONITRING.ACTIVE
CALL OP_Alarm_Monitor : Op_Alarm_Monitor (Alm_Monitor_1 := MAIN_PWR_ERR, Alm_Monitor_2 := W0.02, Alm_Monitor_3 := H16.14, Alm_Monitor_4 := P_Off, Alm_Monitor_5 := P_Off, Alm_Monitor_6 := P_Off, Alm_Monitor_7 := MC_LONG_AXIS_ERR, Alm_Monitor_8 := MC_VERT_AXIS_ERR, Alm_Monitor_9 := MC_TRANS_AXIS_ERR, Alm_Monitor_10 := H13.15, Alm_Monitor_11 := H14.14, Alm_Monitor_12 := P_Off, Alm_Monitor_13 := P_Off, Alm_Monitor_14 := P_Off, Alm_Monitor_15 := P_Off, Alm_Monitor_16 := P_Off, Alarm_State => OP_ALARM_STATE_ACTIVE)  ; MAIN.POWER.ERR, W0.11, RECIPE.ERROR, LONG.AXIS.ERROR.EXISTS, MC.VERTICAL.AXIS.ERROR, TRANSVERSE.AXIS.ERROR.EXISTS, OP.ALARM.SAW.SOFT.START.FAULTED, OP.ALARM.WATER.FLOW.ERROR, OP.ALARM.STATE.ACTIVE(FAULTED)
OUT OP_ALM_MON_EN  ; OP.ALARM.MONITORING.ENABLED
; rung 2
LD OP_ALARM_STATE_ACTIVE  ; OP.ALARM.STATE.ACTIVE(FAULTED)
OUT OI_ALM_IND  ; OI.ALARM.INDICATOR.ACTIVE
; rung 3
LD W121.09  ; OI.ALARM.ACCEPT.CONFIRMATION
OR OI_CTL_ALM_RESET  ; OPERATION.CONTROL.ALARM.RESET.PB
OUT H0.11  ; OPERATION.ALARM.RESET.COMMAND
; rung 4
@LDNOT OP_ALARM_STATE_ACTIVE  ; OP.ALARM.STATE.ACTIVE(FAULTED)
RSET W121.09  ; OI.ALARM.ACCEPT.CONFIRMATION

### Section Ctl_Power

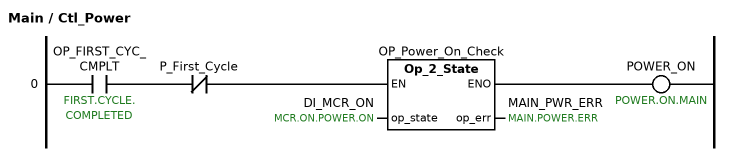
; rung 0
LD OP_FIRST_CYC_CMPLT  ; FIRST.CYCLE.COMPLETED
ANDNOT P_First_Cycle
CALL OP_Power_On_Check : Op_2_State (op_state := DI_MCR_ON, op_err => MAIN_PWR_ERR)  ; MCR.ON.POWER.ON, MAIN.POWER.ERR
OUT POWER_ON  ; POWER.ON.MAIN

### Section Ctl_Safety

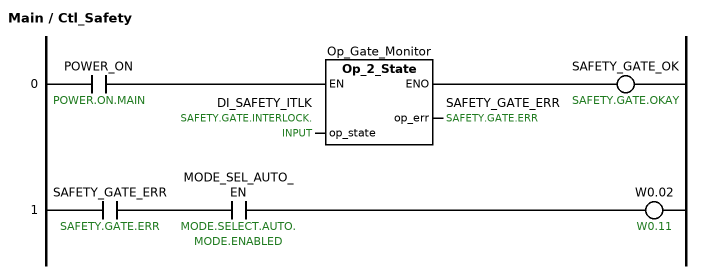
; rung 0
LD POWER_ON  ; POWER.ON.MAIN
CALL Op_Gate_Monitor : Op_2_State (op_state := DI_SAFETY_ITLK, op_err => SAFETY_GATE_ERR)  ; SAFETY.GATE.INTERLOCK.INPUT, SAFETY.GATE.ERR
OUT SAFETY_GATE_OK  ; SAFETY.GATE.OKAY
; rung 1
LD SAFETY_GATE_ERR  ; SAFETY.GATE.ERR
AND MODE_SEL_AUTO_EN  ; MODE.SELECT.AUTO.MODE.ENABLED
OUT W0.02  ; W0.11

### Section Ctl_Mode

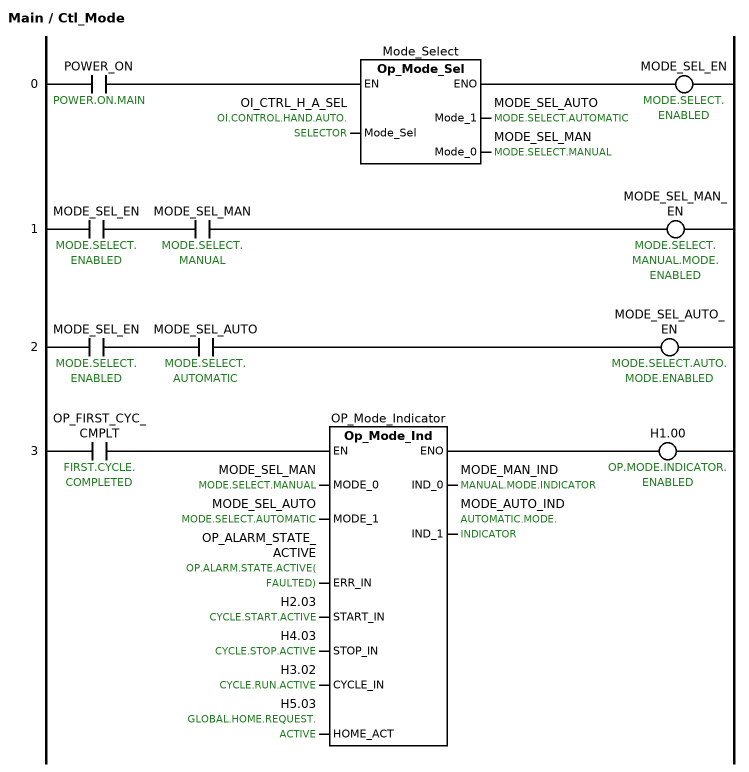
; rung 0
LD POWER_ON  ; POWER.ON.MAIN
CALL Mode_Select : Op_Mode_Sel (Mode_Sel := OI_CTRL_H_A_SEL, Mode_1 => MODE_SEL_AUTO, Mode_0 => MODE_SEL_MAN)  ; OI.CONTROL.HAND.AUTO.SELECTOR, MODE.SELECT.AUTOMATIC, MODE.SELECT.MANUAL
OUT MODE_SEL_EN  ; MODE.SELECT.ENABLED
; rung 1
LD MODE_SEL_EN  ; MODE.SELECT.ENABLED
AND MODE_SEL_MAN  ; MODE.SELECT.MANUAL
OUT MODE_SEL_MAN_EN  ; MODE.SELECT.MANUAL.MODE.ENABLED
; rung 2
LD MODE_SEL_EN  ; MODE.SELECT.ENABLED
AND MODE_SEL_AUTO  ; MODE.SELECT.AUTOMATIC
OUT MODE_SEL_AUTO_EN  ; MODE.SELECT.AUTO.MODE.ENABLED
; rung 3
LD OP_FIRST_CYC_CMPLT  ; FIRST.CYCLE.COMPLETED
CALL OP_Mode_Indicator : Op_Mode_Ind (MODE_0 := MODE_SEL_MAN, MODE_1 := MODE_SEL_AUTO, ERR_IN := OP_ALARM_STATE_ACTIVE, START_IN := H2.03, STOP_IN := H4.03, CYCLE_IN := H3.02, HOME_ACT := H5.03, IND_0 => MODE_MAN_IND, IND_1 => MODE_AUTO_IND)  ; MODE.SELECT.MANUAL, MODE.SELECT.AUTOMATIC, OP.ALARM.STATE.ACTIVE(FAULTED), CYCLE.START.ACTIVE, CYCLE.STOP.ACTIVE, CYCLE.RUN.ACTIVE, GLOBAL.HOME.REQUEST.ACTIVE, MANUAL.MODE.INDICATOR, AUTOMATIC.MODE.INDICATOR
OUT H1.00  ; OP.MODE.INDICATOR.ENABLED

### Section Ctl_Cycle_Start

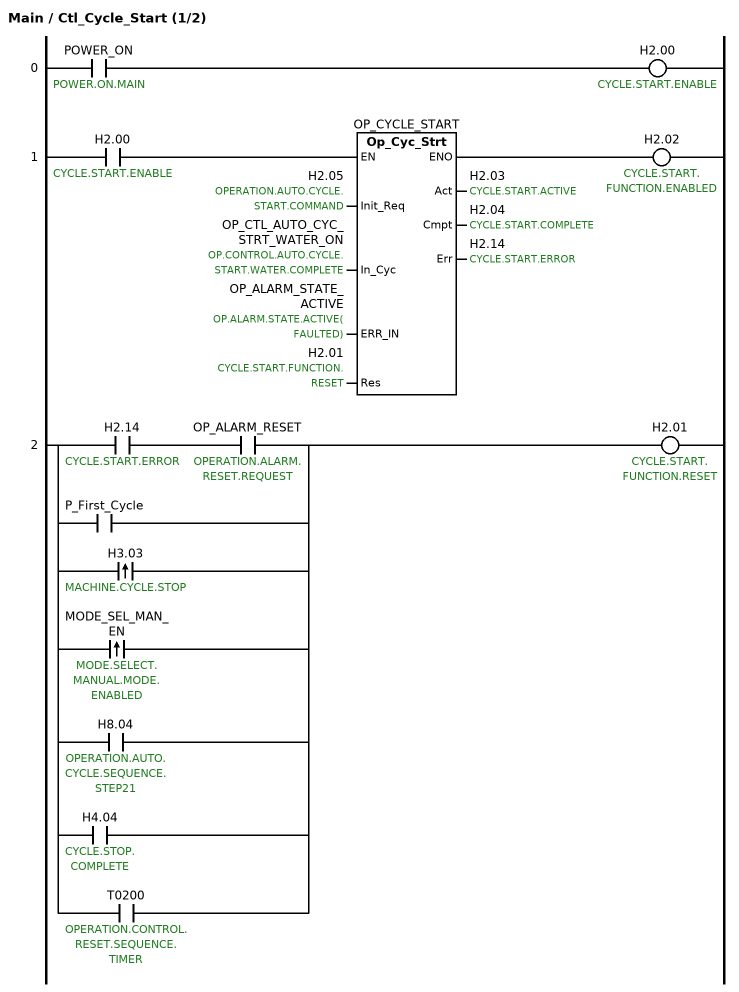
; rung 0
LD POWER_ON  ; POWER.ON.MAIN
OUT H2.00  ; CYCLE.START.ENABLE
; rung 1
LD H2.00  ; CYCLE.START.ENABLE
CALL OP_CYCLE_START : Op_Cyc_Strt (Init_Req := H2.05, In_Cyc := OP_CTL_AUTO_CYC_STRT_WATER_ON, ERR_IN := OP_ALARM_STATE_ACTIVE, Res := H2.01, Act => H2.03, Cmpt => H2.04, Err => H2.14)  ; OPERATION.AUTO.CYCLE.START.COMMAND, OP.CONTROL.AUTO.CYCLE.START.WATER.COMPLETE, OP.ALARM.STATE.ACTIVE(FAULTED), CYCLE.START.FUNCTION.RESET, CYCLE.START.ACTIVE, CYCLE.START.COMPLETE, CYCLE.START.ERROR
OUT H2.02  ; CYCLE.START.FUNCTION.ENABLED
; rung 2
LD H2.14  ; CYCLE.START.ERROR
AND OP_ALARM_RESET  ; OPERATION.ALARM.RESET.REQUEST
OR P_First_Cycle
@OR H3.03  ; MACHINE.CYCLE.STOP
@OR MODE_SEL_MAN_EN  ; MODE.SELECT.MANUAL.MODE.ENABLED
OR H8.04  ; OPERATION.AUTO.CYCLE.SEQUENCE.STEP21
OR H4.04  ; CYCLE.STOP.COMPLETE
OR T0200  ; OPERATION.CONTROL.RESET.SEQUENCE.TIMER
OUT H2.01  ; CYCLE.START.FUNCTION.RESET

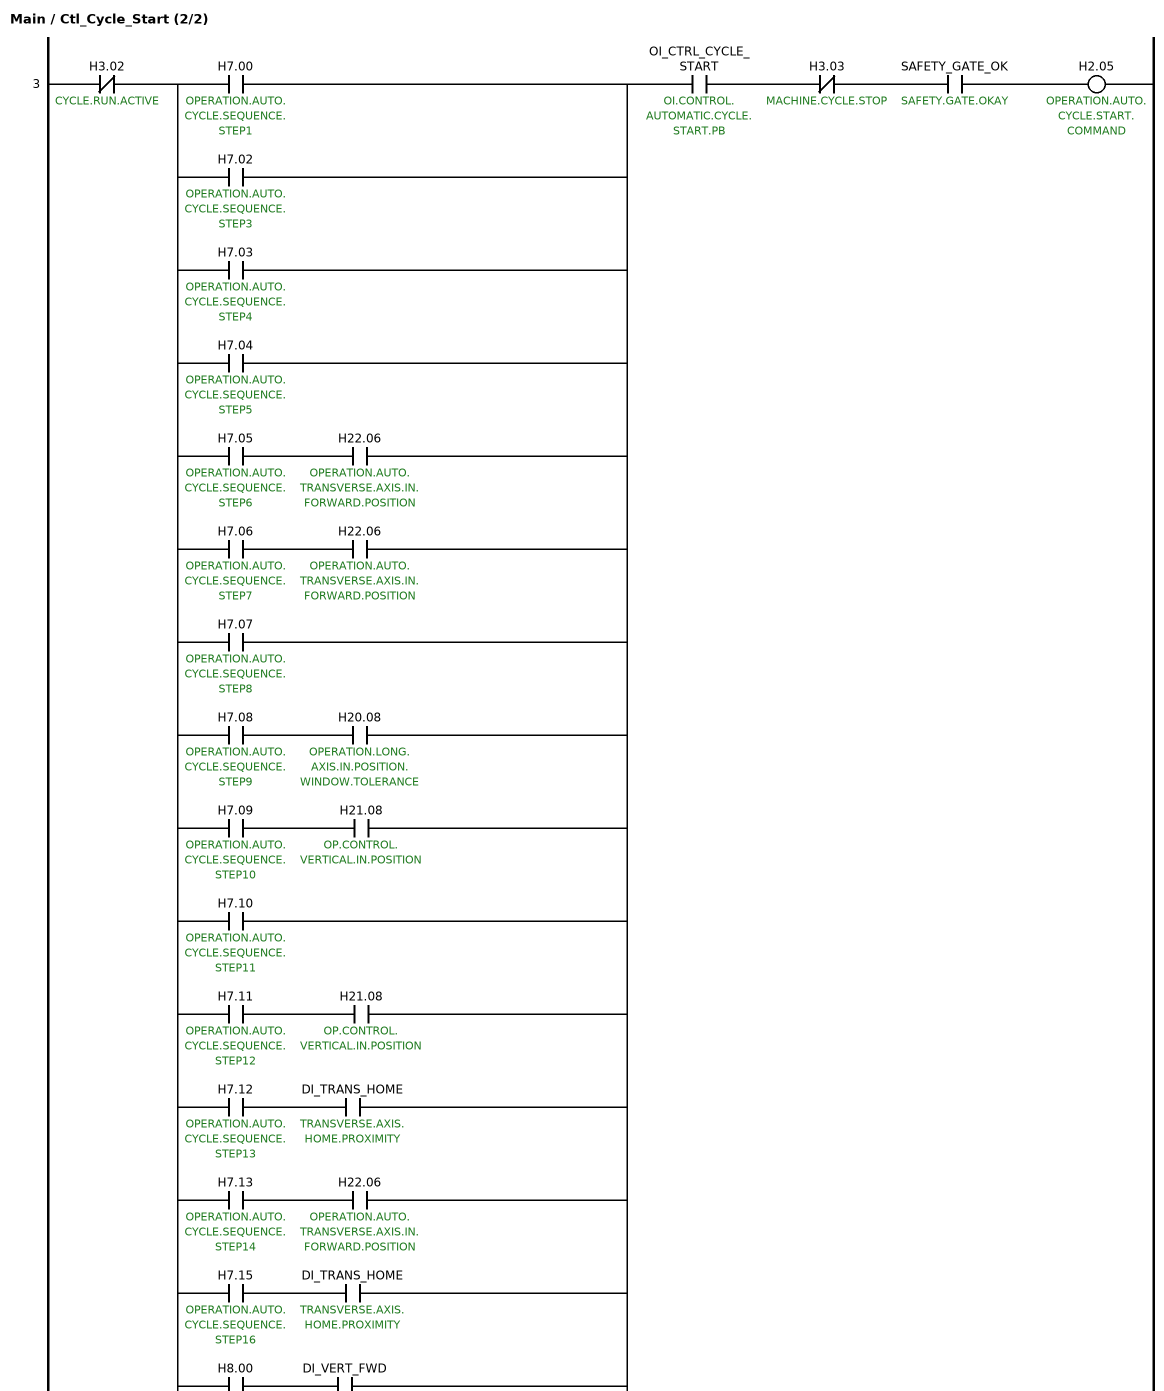

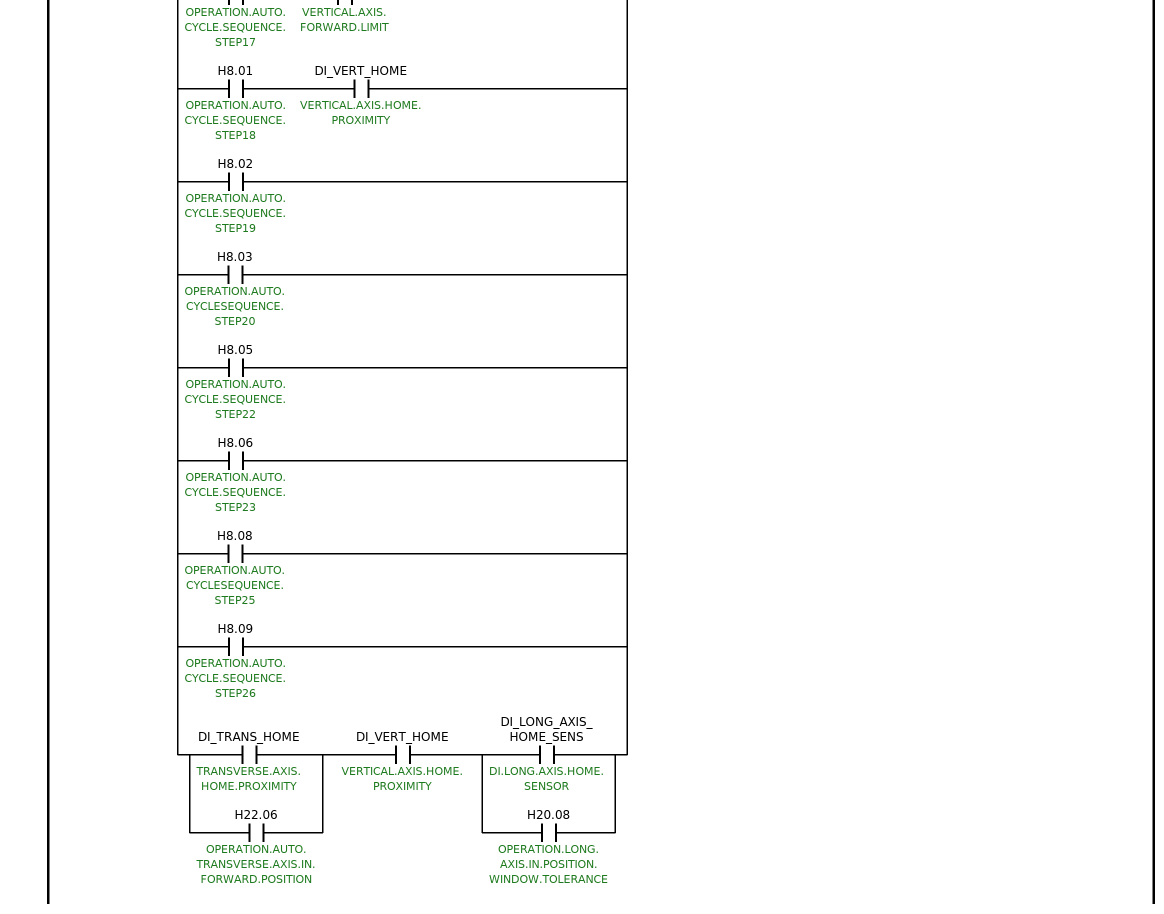
; rung 3
LDNOT H3.02  ; CYCLE.RUN.ACTIVE
LD H7.00  ; OPERATION.AUTO.CYCLE.SEQUENCE.STEP1
OR H7.02  ; OPERATION.AUTO.CYCLE.SEQUENCE.STEP3
OR H7.03  ; OPERATION.AUTO.CYCLE.SEQUENCE.STEP4
OR H7.04  ; OPERATION.AUTO.CYCLE.SEQUENCE.STEP5
LD H7.05  ; OPERATION.AUTO.CYCLE.SEQUENCE.STEP6
AND H22.06  ; OPERATION.AUTO.TRANSVERSE.AXIS.IN.FORWARD.POSITION
ORLD
LD H7.06  ; OPERATION.AUTO.CYCLE.SEQUENCE.STEP7
AND H22.06  ; OPERATION.AUTO.TRANSVERSE.AXIS.IN.FORWARD.POSITION
ORLD
OR H7.07  ; OPERATION.AUTO.CYCLE.SEQUENCE.STEP8
LD H7.08  ; OPERATION.AUTO.CYCLE.SEQUENCE.STEP9
AND H20.08  ; OPERATION.LONG.AXIS.IN.POSITION.WINDOW.TOLERANCE
ORLD
LD H7.09  ; OPERATION.AUTO.CYCLE.SEQUENCE.STEP10
AND H21.08  ; OP.CONTROL.VERTICAL.IN.POSITION
ORLD
OR H7.10  ; OPERATION.AUTO.CYCLE.SEQUENCE.STEP11
LD H7.11  ; OPERATION.AUTO.CYCLE.SEQUENCE.STEP12
AND H21.08  ; OP.CONTROL.VERTICAL.IN.POSITION
ORLD
LD H7.12  ; OPERATION.AUTO.CYCLE.SEQUENCE.STEP13
AND DI_TRANS_HOME  ; TRANSVERSE.AXIS.HOME.PROXIMITY
ORLD
LD H7.13  ; OPERATION.AUTO.CYCLE.SEQUENCE.STEP14
AND H22.06  ; OPERATION.AUTO.TRANSVERSE.AXIS.IN.FORWARD.POSITION
ORLD
LD H7.15  ; OPERATION.AUTO.CYCLE.SEQUENCE.STEP16
AND DI_TRANS_HOME  ; TRANSVERSE.AXIS.HOME.PROXIMITY
ORLD
LD H8.00  ; OPERATION.AUTO.CYCLE.SEQUENCE.STEP17
AND DI_VERT_FWD  ; VERTICAL.AXIS.FORWARD.LIMIT
ORLD
LD H8.01  ; OPERATION.AUTO.CYCLE.SEQUENCE.STEP18
AND DI_VERT_HOME  ; VERTICAL.AXIS.HOME.PROXIMITY
ORLD
OR H8.02  ; OPERATION.AUTO.CYCLE.SEQUENCE.STEP19
OR H8.03  ; OPERATION.AUTO.CYCLESEQUENCE.STEP20
OR H8.05  ; OPERATION.AUTO.CYCLE.SEQUENCE.STEP22
OR H8.06  ; OPERATION.AUTO.CYCLE.SEQUENCE.STEP23
OR H8.08  ; OPERATION.AUTO.CYCLESEQUENCE.STEP25
OR H8.09  ; OPERATION.AUTO.CYCLE.SEQUENCE.STEP26
LD DI_TRANS_HOME  ; TRANSVERSE.AXIS.HOME.PROXIMITY
OR H22.06  ; OPERATION.AUTO.TRANSVERSE.AXIS.IN.FORWARD.POSITION
AND DI_VERT_HOME  ; VERTICAL.AXIS.HOME.PROXIMITY
LD DI_LONG_AXIS_HOME_SENS  ; DI.LONG.AXIS.HOME.SENSOR
OR H20.08  ; OPERATION.LONG.AXIS.IN.POSITION.WINDOW.TOLERANCE
ANDLD
ORLD
ANDLD
AND OI_CTRL_CYCLE_START  ; OI.CONTROL.AUTOMATIC.CYCLE.START.PB
ANDNOT H3.03  ; MACHINE.CYCLE.STOP
AND SAFETY_GATE_OK  ; SAFETY.GATE.OKAY
OUT H2.05  ; OPERATION.AUTO.CYCLE.START.COMMAND

### Section Ctl_Cycle_Run

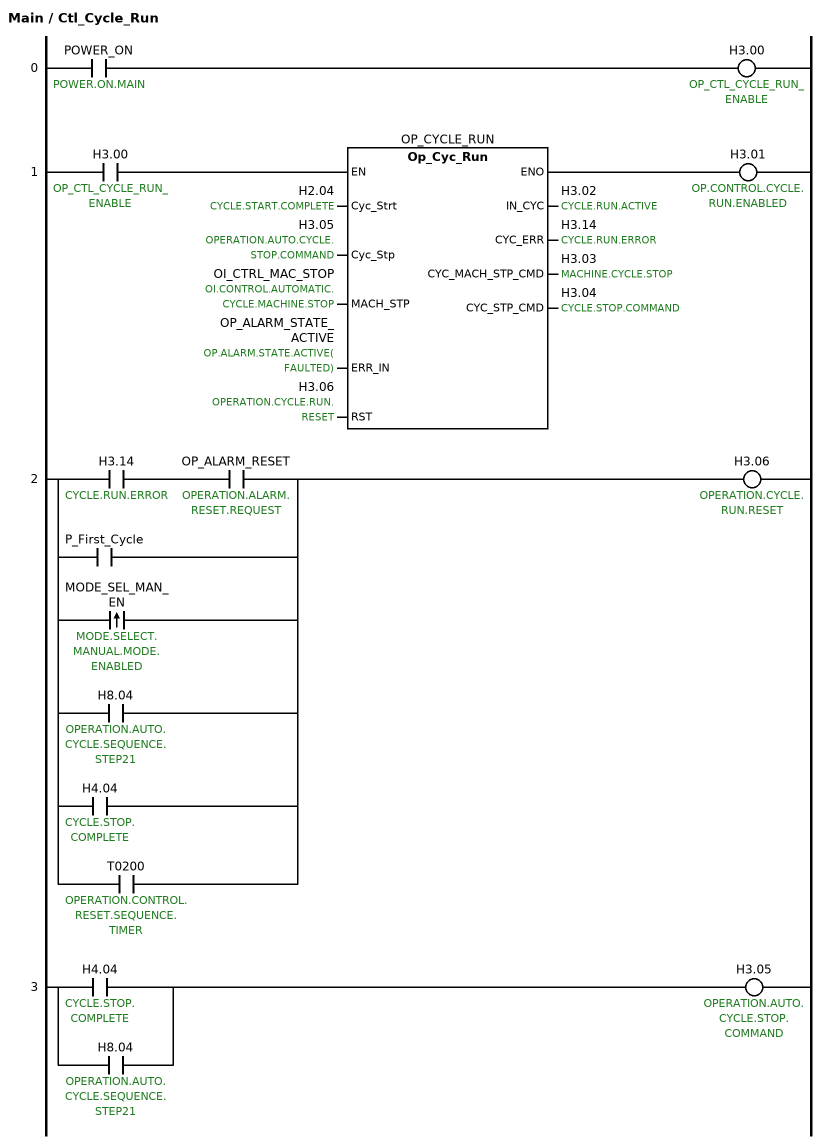
; rung 0
LD POWER_ON  ; POWER.ON.MAIN
OUT H3.00  ; OP_CTL_CYCLE_RUN_ENABLE
; rung 1
LD H3.00  ; OP_CTL_CYCLE_RUN_ENABLE
CALL OP_CYCLE_RUN : Op_Cyc_Run (Cyc_Strt := H2.04, Cyc_Stp := H3.05, MACH_STP := OI_CTRL_MAC_STOP, ERR_IN := OP_ALARM_STATE_ACTIVE, RST := H3.06, IN_CYC => H3.02, CYC_ERR => H3.14, CYC_MACH_STP_CMD => H3.03, CYC_STP_CMD => H3.04)  ; CYCLE.START.COMPLETE, OPERATION.AUTO.CYCLE.STOP.COMMAND, OI.CONTROL.AUTOMATIC.CYCLE.MACHINE.STOP, OP.ALARM.STATE.ACTIVE(FAULTED), OPERATION.CYCLE.RUN.RESET, CYCLE.RUN.ACTIVE, CYCLE.RUN.ERROR, MACHINE.CYCLE.STOP, CYCLE.STOP.COMMAND
OUT H3.01  ; OP.CONTROL.CYCLE.RUN.ENABLED
; rung 2
LD H3.14  ; CYCLE.RUN.ERROR
AND OP_ALARM_RESET  ; OPERATION.ALARM.RESET.REQUEST
OR P_First_Cycle
@OR MODE_SEL_MAN_EN  ; MODE.SELECT.MANUAL.MODE.ENABLED
OR H8.04  ; OPERATION.AUTO.CYCLE.SEQUENCE.STEP21
OR H4.04  ; CYCLE.STOP.COMPLETE
OR T0200  ; OPERATION.CONTROL.RESET.SEQUENCE.TIMER
OUT H3.06  ; OPERATION.CYCLE.RUN.RESET
; rung 3
LD H4.04  ; CYCLE.STOP.COMPLETE
OR H8.04  ; OPERATION.AUTO.CYCLE.SEQUENCE.STEP21
OUT H3.05  ; OPERATION.AUTO.CYCLE.STOP.COMMAND

### Section Ctl_Cycle_Stop

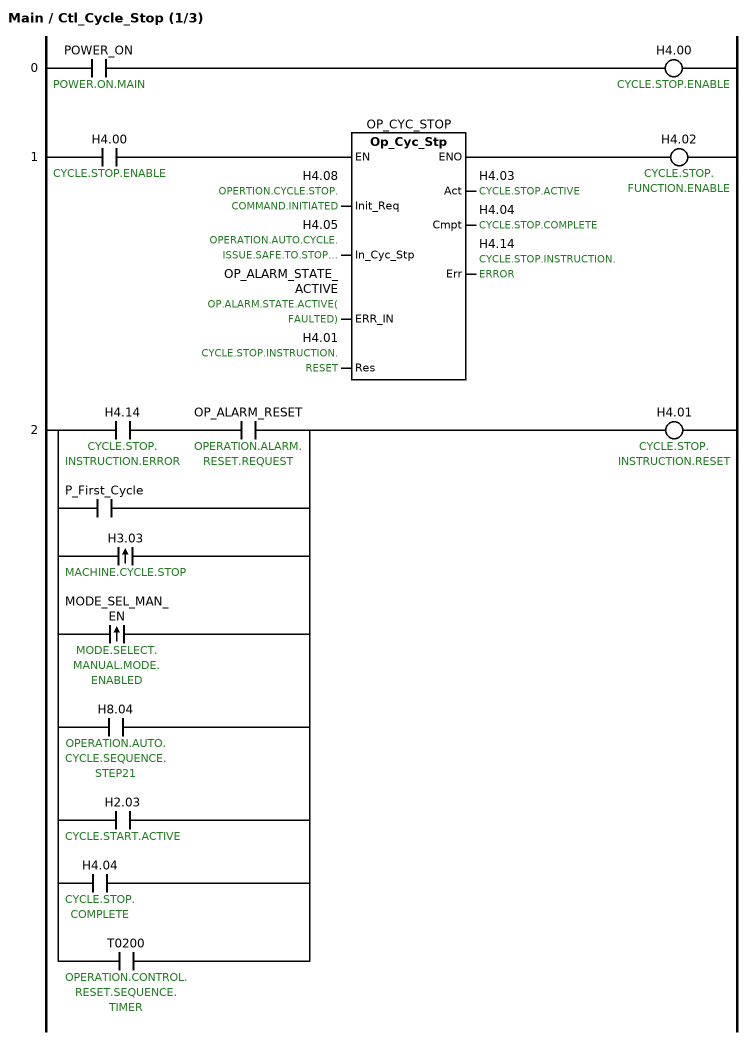
; rung 0
LD POWER_ON  ; POWER.ON.MAIN
OUT H4.00  ; CYCLE.STOP.ENABLE
; rung 1
LD H4.00  ; CYCLE.STOP.ENABLE
CALL OP_CYC_STOP : Op_Cyc_Stp (Init_Req := H4.08, In_Cyc_Stp := H4.05, ERR_IN := OP_ALARM_STATE_ACTIVE, Res := H4.01, Act => H4.03, Cmpt => H4.04, Err => H4.14)  ; OPERTION.CYCLE.STOP.COMMAND.INITIATED, OPERATION.AUTO.CYCLE.ISSUE.SAFE.TO.STOP.COMMAND, OP.ALARM.STATE.ACTIVE(FAULTED), CYCLE.STOP.INSTRUCTION.RESET, CYCLE.STOP.ACTIVE, CYCLE.STOP.COMPLETE, CYCLE.STOP.INSTRUCTION.ERROR
OUT H4.02  ; CYCLE.STOP.FUNCTION.ENABLE
; rung 2
LD H4.14  ; CYCLE.STOP.INSTRUCTION.ERROR
AND OP_ALARM_RESET  ; OPERATION.ALARM.RESET.REQUEST
OR P_First_Cycle
@OR H3.03  ; MACHINE.CYCLE.STOP
@OR MODE_SEL_MAN_EN  ; MODE.SELECT.MANUAL.MODE.ENABLED
OR H8.04  ; OPERATION.AUTO.CYCLE.SEQUENCE.STEP21
OR H2.03  ; CYCLE.START.ACTIVE
OR H4.04  ; CYCLE.STOP.COMPLETE
OR T0200  ; OPERATION.CONTROL.RESET.SEQUENCE.TIMER
OUT H4.01  ; CYCLE.STOP.INSTRUCTION.RESET

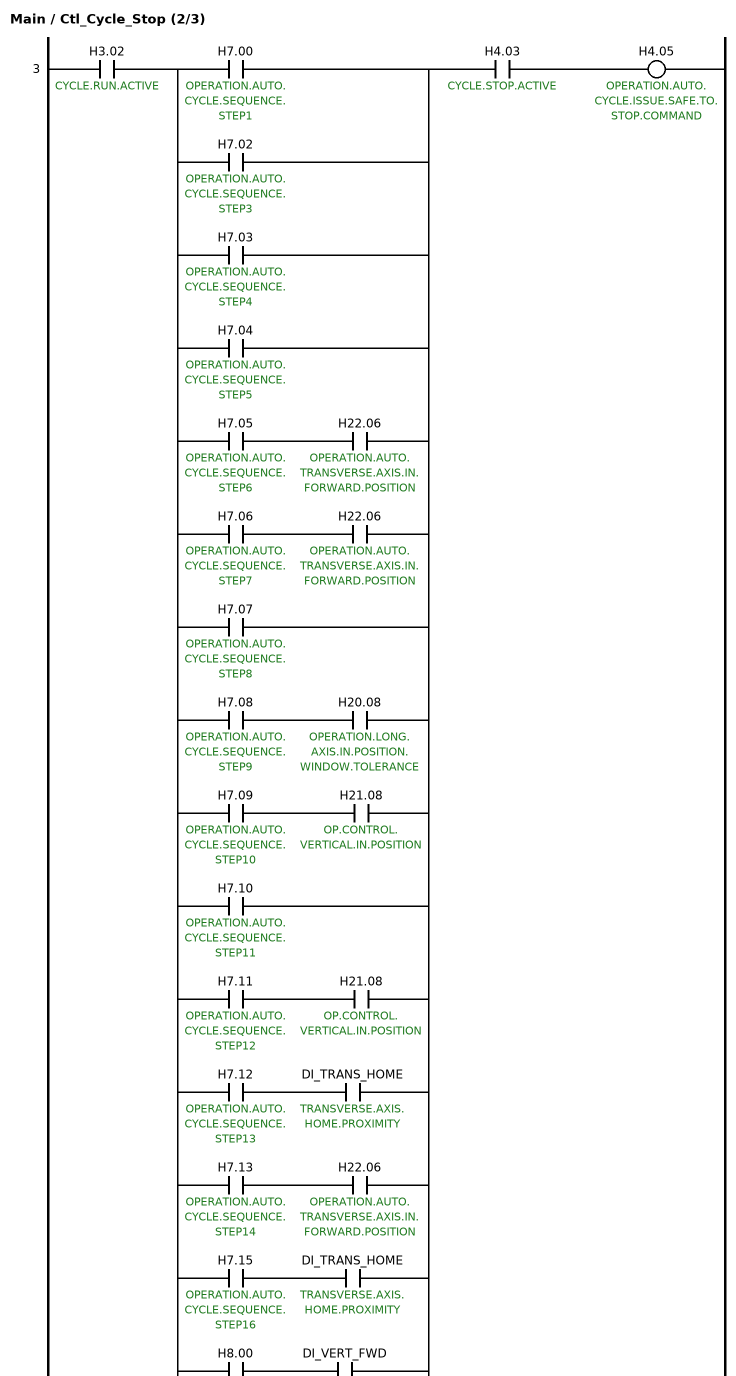

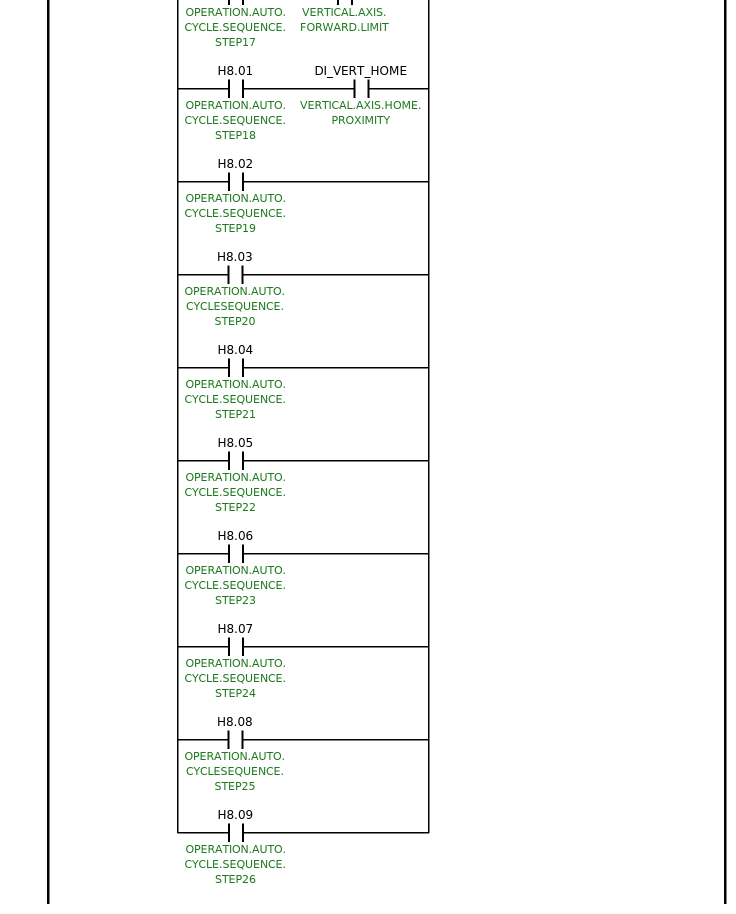
; rung 3
LD H3.02  ; CYCLE.RUN.ACTIVE
LD H7.00  ; OPERATION.AUTO.CYCLE.SEQUENCE.STEP1
OR H7.02  ; OPERATION.AUTO.CYCLE.SEQUENCE.STEP3
OR H7.03  ; OPERATION.AUTO.CYCLE.SEQUENCE.STEP4
OR H7.04  ; OPERATION.AUTO.CYCLE.SEQUENCE.STEP5
LD H7.05  ; OPERATION.AUTO.CYCLE.SEQUENCE.STEP6
AND H22.06  ; OPERATION.AUTO.TRANSVERSE.AXIS.IN.FORWARD.POSITION
ORLD
LD H7.06  ; OPERATION.AUTO.CYCLE.SEQUENCE.STEP7
AND H22.06  ; OPERATION.AUTO.TRANSVERSE.AXIS.IN.FORWARD.POSITION
ORLD
OR H7.07  ; OPERATION.AUTO.CYCLE.SEQUENCE.STEP8
LD H7.08  ; OPERATION.AUTO.CYCLE.SEQUENCE.STEP9
AND H20.08  ; OPERATION.LONG.AXIS.IN.POSITION.WINDOW.TOLERANCE
ORLD
LD H7.09  ; OPERATION.AUTO.CYCLE.SEQUENCE.STEP10
AND H21.08  ; OP.CONTROL.VERTICAL.IN.POSITION
ORLD
OR H7.10  ; OPERATION.AUTO.CYCLE.SEQUENCE.STEP11
LD H7.11  ; OPERATION.AUTO.CYCLE.SEQUENCE.STEP12
AND H21.08  ; OP.CONTROL.VERTICAL.IN.POSITION
ORLD
LD H7.12  ; OPERATION.AUTO.CYCLE.SEQUENCE.STEP13
AND DI_TRANS_HOME  ; TRANSVERSE.AXIS.HOME.PROXIMITY
ORLD
LD H7.13  ; OPERATION.AUTO.CYCLE.SEQUENCE.STEP14
AND H22.06  ; OPERATION.AUTO.TRANSVERSE.AXIS.IN.FORWARD.POSITION
ORLD
LD H7.15  ; OPERATION.AUTO.CYCLE.SEQUENCE.STEP16
AND DI_TRANS_HOME  ; TRANSVERSE.AXIS.HOME.PROXIMITY
ORLD
LD H8.00  ; OPERATION.AUTO.CYCLE.SEQUENCE.STEP17
AND DI_VERT_FWD  ; VERTICAL.AXIS.FORWARD.LIMIT
ORLD
LD H8.01  ; OPERATION.AUTO.CYCLE.SEQUENCE.STEP18
AND DI_VERT_HOME  ; VERTICAL.AXIS.HOME.PROXIMITY
ORLD
OR H8.02  ; OPERATION.AUTO.CYCLE.SEQUENCE.STEP19
OR H8.03  ; OPERATION.AUTO.CYCLESEQUENCE.STEP20
OR H8.04  ; OPERATION.AUTO.CYCLE.SEQUENCE.STEP21
OR H8.05  ; OPERATION.AUTO.CYCLE.SEQUENCE.STEP22
OR H8.06  ; OPERATION.AUTO.CYCLE.SEQUENCE.STEP23
OR H8.07  ; OPERATION.AUTO.CYCLE.SEQUENCE.STEP24
OR H8.08  ; OPERATION.AUTO.CYCLESEQUENCE.STEP25
OR H8.09  ; OPERATION.AUTO.CYCLE.SEQUENCE.STEP26
ANDLD
AND H4.03  ; CYCLE.STOP.ACTIVE
OUT H4.05  ; OPERATION.AUTO.CYCLE.ISSUE.SAFE.TO.STOP.COMMAND

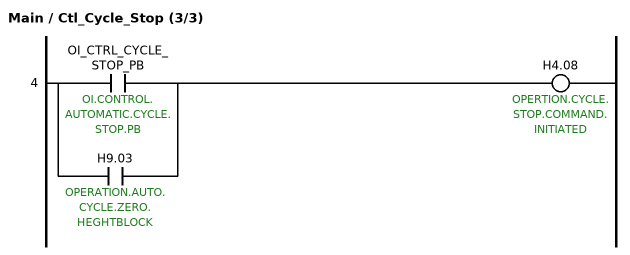
; rung 4
LD OI_CTRL_CYCLE_STOP_PB  ; OI.CONTROL.AUTOMATIC.CYCLE.STOP.PB
OR H9.03  ; OPERATION.AUTO.CYCLE.ZERO.HEGHTBLOCK
OUT H4.08  ; OPERTION.CYCLE.STOP.COMMAND.INITIATED

### Section Ctl_Auto_Cycle_Sequence

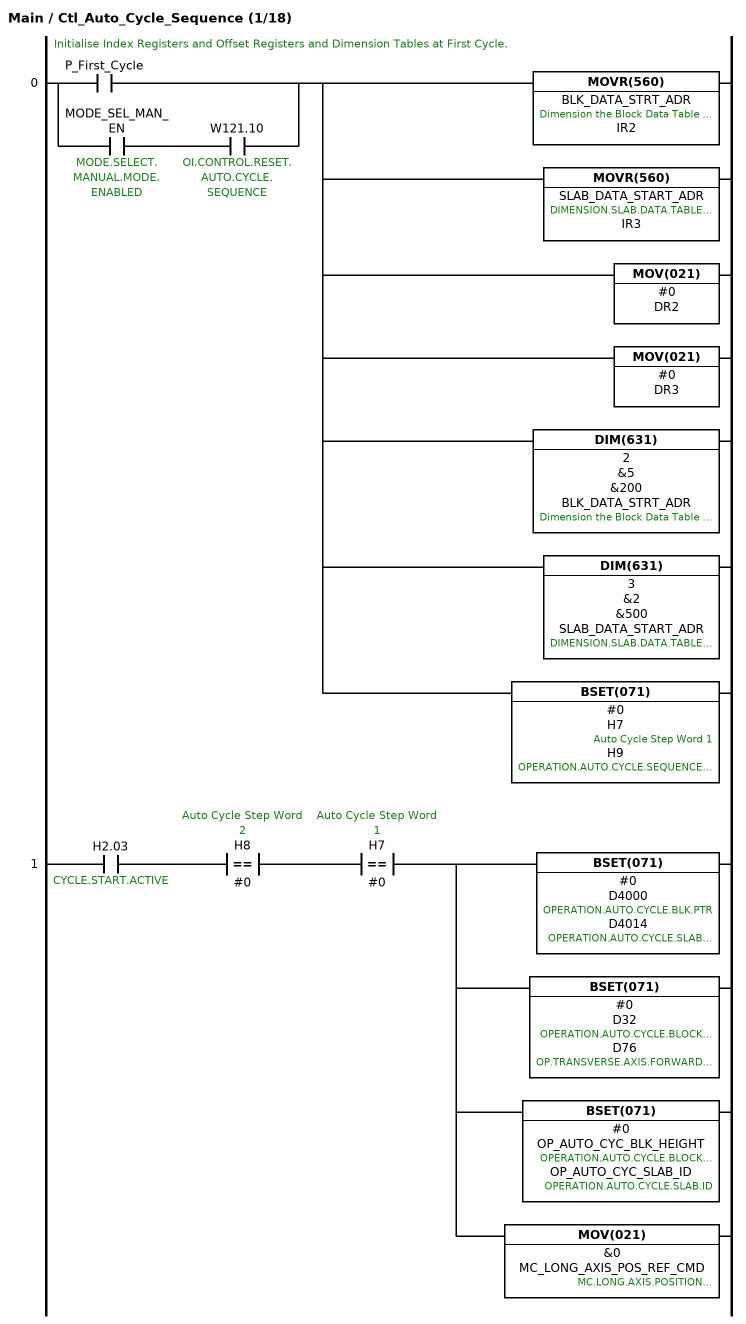
; rung 0: Initialise Index Registers and Offset Registers and Dimension Tables at First Cycle.
LD P_First_Cycle
LD MODE_SEL_MAN_EN  ; MODE.SELECT.MANUAL.MODE.ENABLED
AND W121.10  ; OI.CONTROL.RESET.AUTO.CYCLE.SEQUENCE
ORLD
MOVR(560) BLK_DATA_STRT_ADR IR2  ; Dimension the Block Data Table - Start Address
MOVR(560) SLAB_DATA_START_ADR IR3  ; DIMENSION.SLAB.DATA.TABLE.START.ADDRESS
MOV(021) #0 DR2
MOV(021) #0 DR3
DIM(631) 2 &5 &200 BLK_DATA_STRT_ADR  ; Dimension the Block Data Table - Start Address
DIM(631) 3 &2 &500 SLAB_DATA_START_ADR  ; DIMENSION.SLAB.DATA.TABLE.START.ADDRESS
BSET(071) #0 H7 H9  ; Auto Cycle Step Word 1, OPERATION.AUTO.CYCLE.SEQUENCE.STATE.BITS
; rung 1
LD H2.03  ; CYCLE.START.ACTIVE
AND=(300) H8 #0  ; Auto Cycle Step Word 2
AND=(300) H7 #0  ; Auto Cycle Step Word 1
BSET(071) #0 D4000 D4014  ; OPERATION.AUTO.CYCLE.BLK.PTR, OPERATION.AUTO.CYCLE.SLAB.POINTER
BSET(071) #0 D32 D76  ; OPERATION.AUTO.CYCLE.BLOCK.FIRST.CUT.WORKING.REAL, OP.TRANSVERSE.AXIS.FORWARD.TARGET
BSET(071) #0 OP_AUTO_CYC_BLK_HEIGHT OP_AUTO_CYC_SLAB_ID  ; OPERATION.AUTO.CYCLE.BLOCK.HEIGHT.WORKING, OPERATION.AUTO.CYCLE.SLAB.ID
MOV(021) &0 MC_LONG_AXIS_POS_REF_CMD  ; MC.LONG.AXIS.POSITION.REFERENCE.COMMAND.VALUE

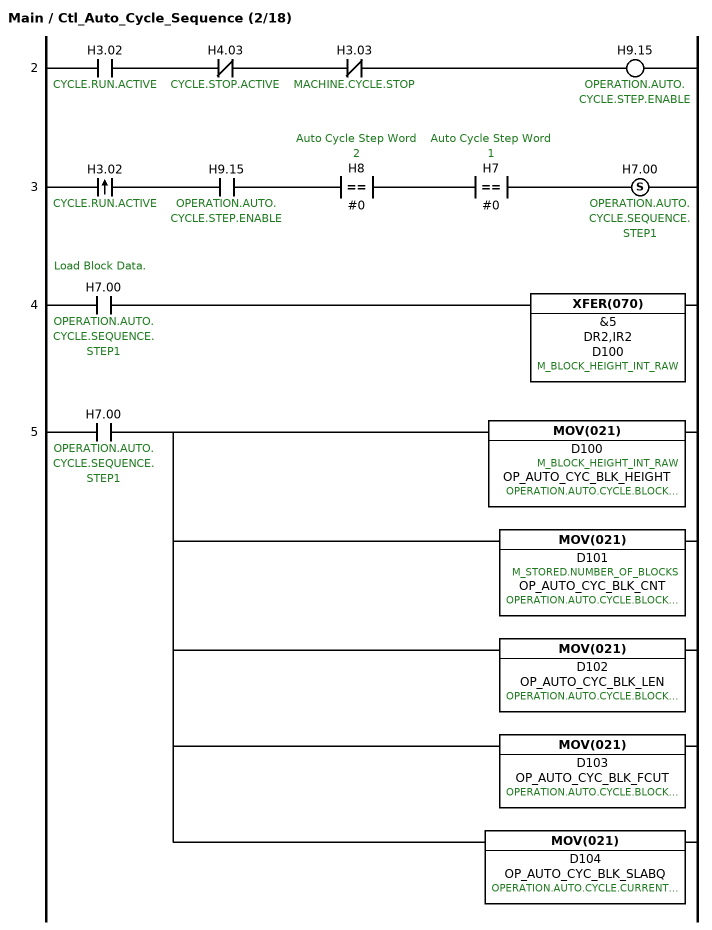
; rung 2
LD H3.02  ; CYCLE.RUN.ACTIVE
ANDNOT H4.03  ; CYCLE.STOP.ACTIVE
ANDNOT H3.03  ; MACHINE.CYCLE.STOP
OUT H9.15  ; OPERATION.AUTO.CYCLE.STEP.ENABLE
; rung 3
@LD H3.02  ; CYCLE.RUN.ACTIVE
AND H9.15  ; OPERATION.AUTO.CYCLE.STEP.ENABLE
AND=(300) H8 #0  ; Auto Cycle Step Word 2
AND=(300) H7 #0  ; Auto Cycle Step Word 1
SET H7.00  ; OPERATION.AUTO.CYCLE.SEQUENCE.STEP1
; rung 4: Load Block Data.
LD H7.00  ; OPERATION.AUTO.CYCLE.SEQUENCE.STEP1
XFER(070) &5 DR2,IR2 D100  ; M_BLOCK_HEIGHT_INT_RAW
; rung 5
LD H7.00  ; OPERATION.AUTO.CYCLE.SEQUENCE.STEP1
MOV(021) D100 OP_AUTO_CYC_BLK_HEIGHT  ; M_BLOCK_HEIGHT_INT_RAW, OPERATION.AUTO.CYCLE.BLOCK.HEIGHT.WORKING
MOV(021) D101 OP_AUTO_CYC_BLK_CNT  ; M_STORED.NUMBER_OF_BLOCKS, OPERATION.AUTO.CYCLE.BLOCK.COUNT
MOV(021) D102 OP_AUTO_CYC_BLK_LEN  ; OPERATION.AUTO.CYCLE.BLOCK.TRANSVERSE.AXIS.STOP.POSITION.WORKING
MOV(021) D103 OP_AUTO_CYC_BLK_FCUT  ; OPERATION.AUTO.CYCLE.BLOCK.FIRST.CUT.WORKING
MOV(021) D104 OP_AUTO_CYC_BLK_SLABQ  ; OPERATION.AUTO.CYCLE.CURRENT.BLOCK.SLAB.QUANTITY

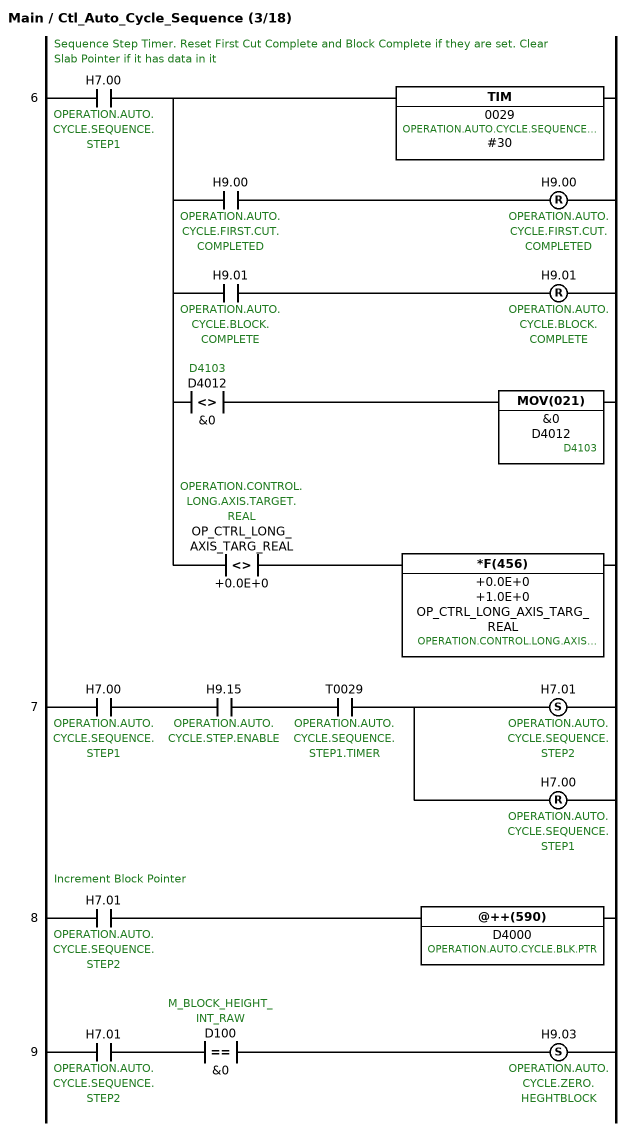
; rung 6: Sequence Step Timer. Reset First Cut Complete and Block Complete if they are set. Clear Slab Pointer if it has data in it
LD H7.00  ; OPERATION.AUTO.CYCLE.SEQUENCE.STEP1
OUT TR0
TIM 0029 #30  ; OPERATION.AUTO.CYCLE.SEQUENCE.STEP1.TIMER
AND H9.00  ; OPERATION.AUTO.CYCLE.FIRST.CUT.COMPLETED
RSET H9.00  ; OPERATION.AUTO.CYCLE.FIRST.CUT.COMPLETED
LD TR0
AND H9.01  ; OPERATION.AUTO.CYCLE.BLOCK.COMPLETE
RSET H9.01  ; OPERATION.AUTO.CYCLE.BLOCK.COMPLETE
LD TR0
AND<>(305) D4012 &0  ; D4103
MOV(021) &0 D4012  ; D4103
LD TR0
AND<>F(330) OP_CTRL_LONG_AXIS_TARG_REAL +0.0E+0  ; OPERATION.CONTROL.LONG.AXIS.TARGET.REAL
*F(456) +0.0E+0 +1.0E+0 OP_CTRL_LONG_AXIS_TARG_REAL  ; OPERATION.CONTROL.LONG.AXIS.TARGET.REAL
; rung 7
LD H7.00  ; OPERATION.AUTO.CYCLE.SEQUENCE.STEP1
AND H9.15  ; OPERATION.AUTO.CYCLE.STEP.ENABLE
AND T0029  ; OPERATION.AUTO.CYCLE.SEQUENCE.STEP1.TIMER
SET H7.01  ; OPERATION.AUTO.CYCLE.SEQUENCE.STEP2
RSET H7.00  ; OPERATION.AUTO.CYCLE.SEQUENCE.STEP1
; rung 8: Increment Block Pointer
LD H7.01  ; OPERATION.AUTO.CYCLE.SEQUENCE.STEP2
@++(590) D4000  ; OPERATION.AUTO.CYCLE.BLK.PTR
; rung 9
LD H7.01  ; OPERATION.AUTO.CYCLE.SEQUENCE.STEP2
AND=(300) D100 &0  ; M_BLOCK_HEIGHT_INT_RAW
SET H9.03  ; OPERATION.AUTO.CYCLE.ZERO.HEGHTBLOCK

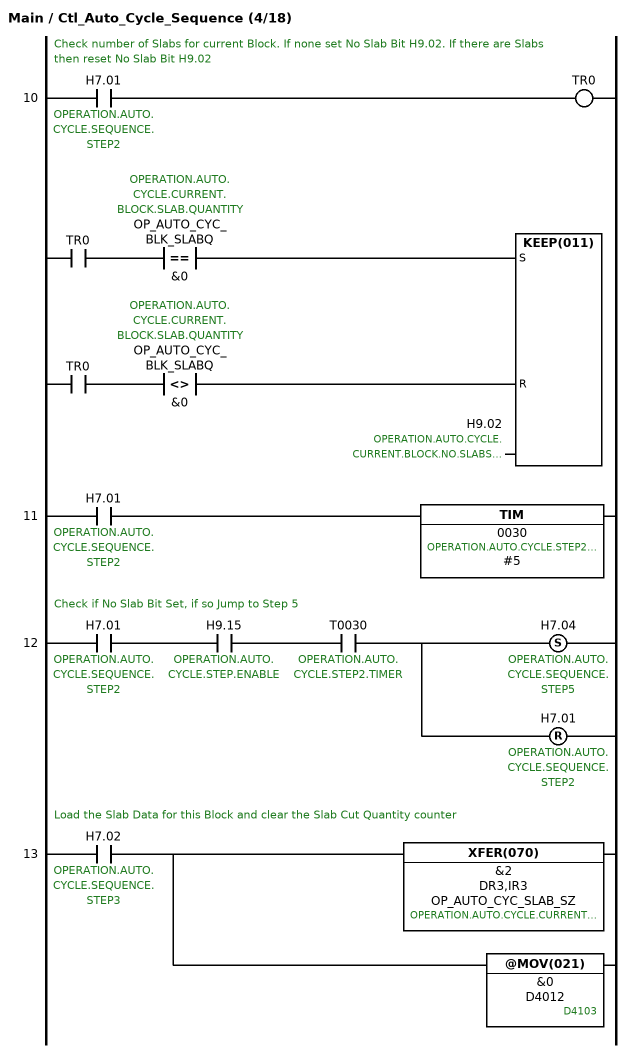
; rung 10: Check number of Slabs for current Block. If none set No Slab Bit H9.02. If there are Slabs then reset No Slab Bit H9.02
LD H7.01  ; OPERATION.AUTO.CYCLE.SEQUENCE.STEP2
OUT TR0
AND=(300) OP_AUTO_CYC_BLK_SLABQ &0  ; OPERATION.AUTO.CYCLE.CURRENT.BLOCK.SLAB.QUANTITY
LD TR0
AND<>(305) OP_AUTO_CYC_BLK_SLABQ &0  ; OPERATION.AUTO.CYCLE.CURRENT.BLOCK.SLAB.QUANTITY
KEEP(011) H9.02  ; OPERATION.AUTO.CYCLE.CURRENT.BLOCK.NO.SLABS.BIT
; rung 11
LD H7.01  ; OPERATION.AUTO.CYCLE.SEQUENCE.STEP2
TIM 0030 #5  ; OPERATION.AUTO.CYCLE.STEP2.TIMER
; rung 12: Check if No Slab Bit Set, if so Jump to Step 5
LD H7.01  ; OPERATION.AUTO.CYCLE.SEQUENCE.STEP2
AND H9.15  ; OPERATION.AUTO.CYCLE.STEP.ENABLE
AND T0030  ; OPERATION.AUTO.CYCLE.STEP2.TIMER
SET H7.04  ; OPERATION.AUTO.CYCLE.SEQUENCE.STEP5
RSET H7.01  ; OPERATION.AUTO.CYCLE.SEQUENCE.STEP2
; rung 13: Load the Slab Data for this Block and clear the Slab Cut Quantity counter
LD H7.02  ; OPERATION.AUTO.CYCLE.SEQUENCE.STEP3
XFER(070) &2 DR3,IR3 OP_AUTO_CYC_SLAB_SZ  ; OPERATION.AUTO.CYCLE.CURRENT.SLAB.SIZE
@MOV(021) &0 D4012  ; D4103

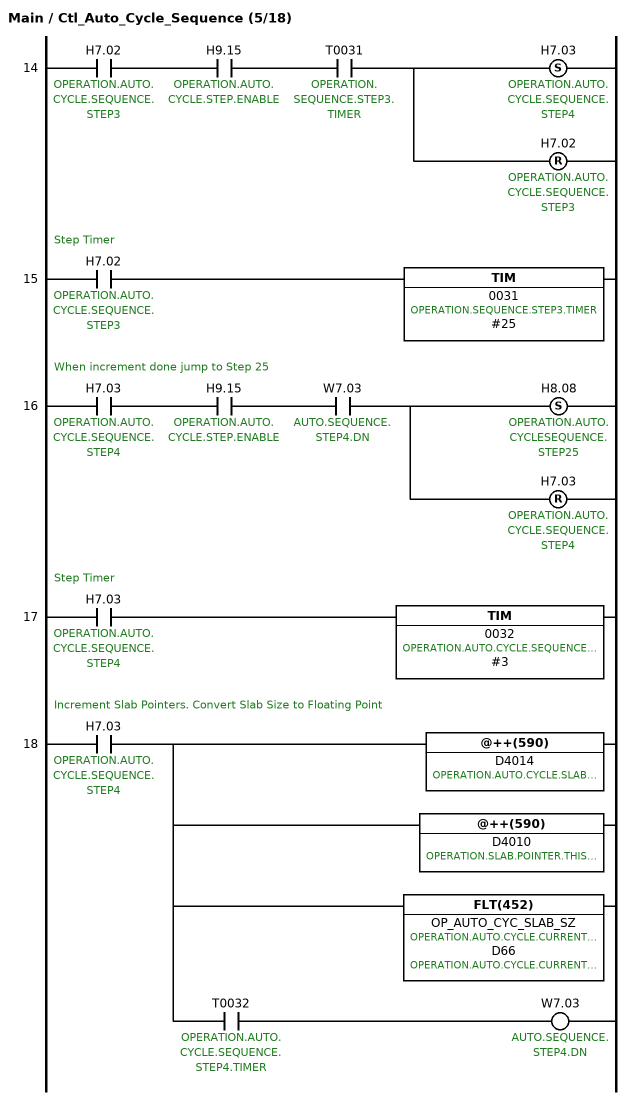
; rung 14
LD H7.02  ; OPERATION.AUTO.CYCLE.SEQUENCE.STEP3
AND H9.15  ; OPERATION.AUTO.CYCLE.STEP.ENABLE
AND T0031  ; OPERATION.SEQUENCE.STEP3.TIMER
SET H7.03  ; OPERATION.AUTO.CYCLE.SEQUENCE.STEP4
RSET H7.02  ; OPERATION.AUTO.CYCLE.SEQUENCE.STEP3
; rung 15: Step Timer
LD H7.02  ; OPERATION.AUTO.CYCLE.SEQUENCE.STEP3
TIM 0031 #25  ; OPERATION.SEQUENCE.STEP3.TIMER
; rung 16: When increment done jump to Step 25
LD H7.03  ; OPERATION.AUTO.CYCLE.SEQUENCE.STEP4
AND H9.15  ; OPERATION.AUTO.CYCLE.STEP.ENABLE
AND W7.03  ; AUTO.SEQUENCE.STEP4.DN
SET H8.08  ; OPERATION.AUTO.CYCLESEQUENCE.STEP25
RSET H7.03  ; OPERATION.AUTO.CYCLE.SEQUENCE.STEP4
; rung 17: Step Timer
LD H7.03  ; OPERATION.AUTO.CYCLE.SEQUENCE.STEP4
TIM 0032 #3  ; OPERATION.AUTO.CYCLE.SEQUENCE.STEP4.TIMER
; rung 18: Increment Slab Pointers. Convert Slab Size to Floating Point
LD H7.03  ; OPERATION.AUTO.CYCLE.SEQUENCE.STEP4
@++(590) D4014  ; OPERATION.AUTO.CYCLE.SLAB.POINTER
@++(590) D4010  ; OPERATION.SLAB.POINTER.THIS.BLOCK
FLT(452) OP_AUTO_CYC_SLAB_SZ D66  ; OPERATION.AUTO.CYCLE.CURRENT.SLAB.SIZE, OPERATION.AUTO.CYCLE.CURRENT.SLAB.SIZE.REAL.RAW
AND T0032  ; OPERATION.AUTO.CYCLE.SEQUENCE.STEP4.TIMER
OUT W7.03  ; AUTO.SEQUENCE.STEP4.DN

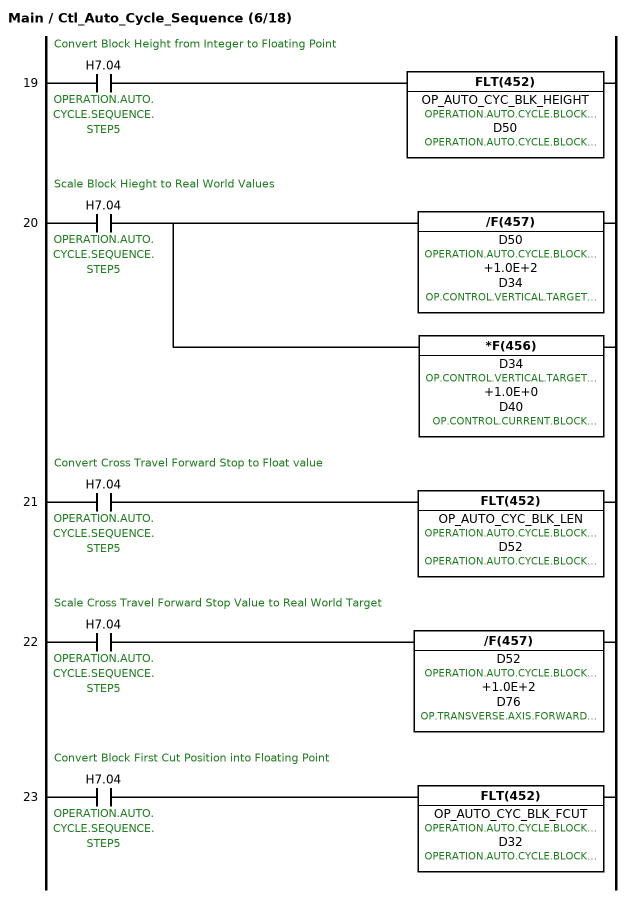
; rung 19: Convert Block Height from Integer to Floating Point
LD H7.04  ; OPERATION.AUTO.CYCLE.SEQUENCE.STEP5
FLT(452) OP_AUTO_CYC_BLK_HEIGHT D50  ; OPERATION.AUTO.CYCLE.BLOCK.HEIGHT.WORKING, OPERATION.AUTO.CYCLE.BLOCK.HEIGHT.REAL
; rung 20: Scale Block Hieght to Real World Values
LD H7.04  ; OPERATION.AUTO.CYCLE.SEQUENCE.STEP5
/F(457) D50 +1.0E+2 D34  ; OPERATION.AUTO.CYCLE.BLOCK.HEIGHT.REAL, OP.CONTROL.VERTICAL.TARGET.SCALED
*F(456) D34 +1.0E+0 D40  ; OP.CONTROL.VERTICAL.TARGET.SCALED, OP.CONTROL.CURRENT.BLOCK.HEIGHT.REAL
; rung 21: Convert Cross Travel Forward Stop to Float value
LD H7.04  ; OPERATION.AUTO.CYCLE.SEQUENCE.STEP5
FLT(452) OP_AUTO_CYC_BLK_LEN D52  ; OPERATION.AUTO.CYCLE.BLOCK.TRANSVERSE.AXIS.STOP.POSITION.WORKING, OPERATION.AUTO.CYCLE.BLOCK.TRANSVERSE.AXIS.FORWARD.STOP.POSITION
; rung 22: Scale Cross Travel Forward Stop Value to Real World Target
LD H7.04  ; OPERATION.AUTO.CYCLE.SEQUENCE.STEP5
/F(457) D52 +1.0E+2 D76  ; OPERATION.AUTO.CYCLE.BLOCK.TRANSVERSE.AXIS.FORWARD.STOP.POSITION, OP.TRANSVERSE.AXIS.FORWARD.TARGET
; rung 23: Convert Block First Cut Position into Floating Point
LD H7.04  ; OPERATION.AUTO.CYCLE.SEQUENCE.STEP5
FLT(452) OP_AUTO_CYC_BLK_FCUT D32  ; OPERATION.AUTO.CYCLE.BLOCK.FIRST.CUT.WORKING, OPERATION.AUTO.CYCLE.BLOCK.FIRST.CUT.WORKING.REAL

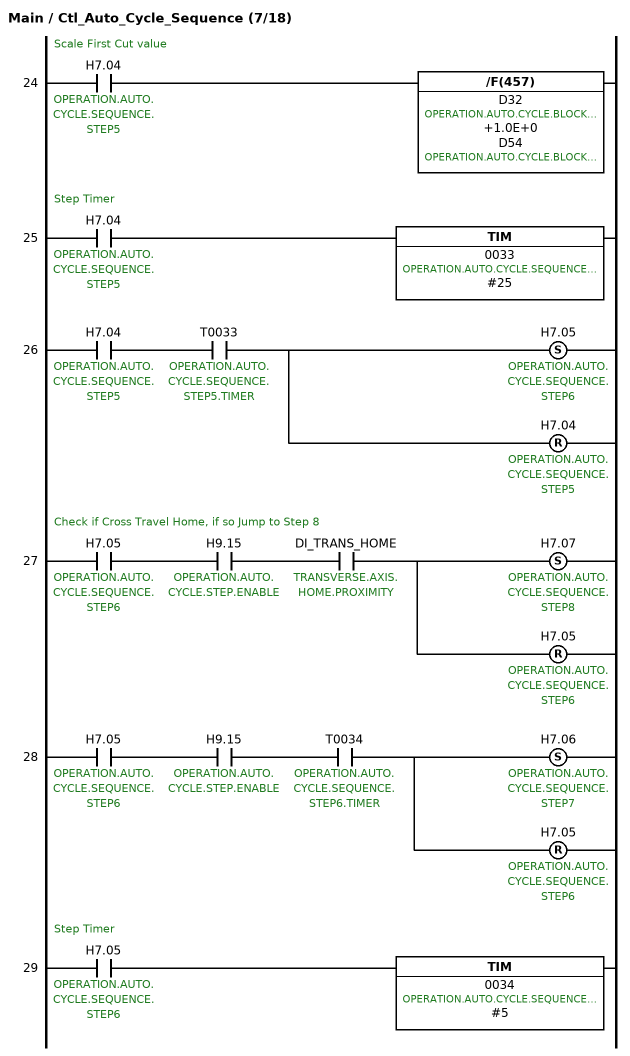
; rung 24: Scale First Cut value
LD H7.04  ; OPERATION.AUTO.CYCLE.SEQUENCE.STEP5
/F(457) D32 +1.0E+0 D54  ; OPERATION.AUTO.CYCLE.BLOCK.FIRST.CUT.WORKING.REAL, OPERATION.AUTO.CYCLE.BLOCK.FIRST.CUT.REAL
; rung 25: Step Timer
LD H7.04  ; OPERATION.AUTO.CYCLE.SEQUENCE.STEP5
TIM 0033 #25  ; OPERATION.AUTO.CYCLE.SEQUENCE.STEP5.TIMER
; rung 26
LD H7.04  ; OPERATION.AUTO.CYCLE.SEQUENCE.STEP5
AND T0033  ; OPERATION.AUTO.CYCLE.SEQUENCE.STEP5.TIMER
SET H7.05  ; OPERATION.AUTO.CYCLE.SEQUENCE.STEP6
RSET H7.04  ; OPERATION.AUTO.CYCLE.SEQUENCE.STEP5
; rung 27: Check if Cross Travel Home, if so Jump to Step 8
LD H7.05  ; OPERATION.AUTO.CYCLE.SEQUENCE.STEP6
AND H9.15  ; OPERATION.AUTO.CYCLE.STEP.ENABLE
AND DI_TRANS_HOME  ; TRANSVERSE.AXIS.HOME.PROXIMITY
SET H7.07  ; OPERATION.AUTO.CYCLE.SEQUENCE.STEP8
RSET H7.05  ; OPERATION.AUTO.CYCLE.SEQUENCE.STEP6
; rung 28
LD H7.05  ; OPERATION.AUTO.CYCLE.SEQUENCE.STEP6
AND H9.15  ; OPERATION.AUTO.CYCLE.STEP.ENABLE
AND T0034  ; OPERATION.AUTO.CYCLE.SEQUENCE.STEP6.TIMER
SET H7.06  ; OPERATION.AUTO.CYCLE.SEQUENCE.STEP7
RSET H7.05  ; OPERATION.AUTO.CYCLE.SEQUENCE.STEP6
; rung 29: Step Timer
LD H7.05  ; OPERATION.AUTO.CYCLE.SEQUENCE.STEP6
TIM 0034 #5  ; OPERATION.AUTO.CYCLE.SEQUENCE.STEP6.TIMER

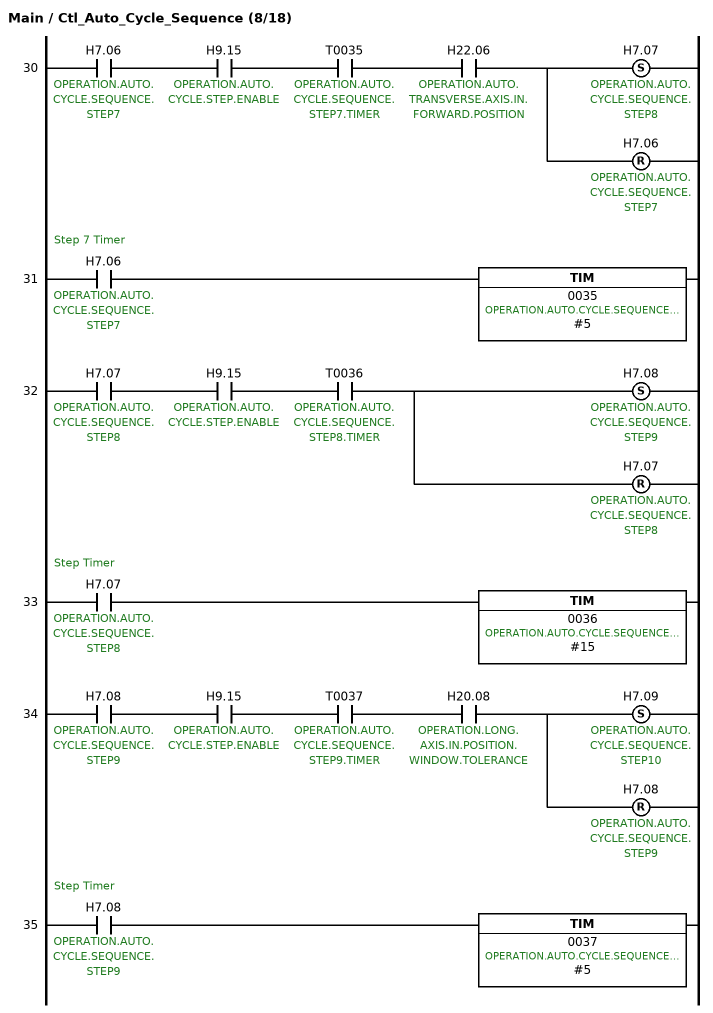
; rung 30
LD H7.06  ; OPERATION.AUTO.CYCLE.SEQUENCE.STEP7
AND H9.15  ; OPERATION.AUTO.CYCLE.STEP.ENABLE
AND T0035  ; OPERATION.AUTO.CYCLE.SEQUENCE.STEP7.TIMER
AND H22.06  ; OPERATION.AUTO.TRANSVERSE.AXIS.IN.FORWARD.POSITION
SET H7.07  ; OPERATION.AUTO.CYCLE.SEQUENCE.STEP8
RSET H7.06  ; OPERATION.AUTO.CYCLE.SEQUENCE.STEP7
; rung 31: Step 7 Timer
LD H7.06  ; OPERATION.AUTO.CYCLE.SEQUENCE.STEP7
TIM 0035 #5  ; OPERATION.AUTO.CYCLE.SEQUENCE.STEP7.TIMER
; rung 32
LD H7.07  ; OPERATION.AUTO.CYCLE.SEQUENCE.STEP8
AND H9.15  ; OPERATION.AUTO.CYCLE.STEP.ENABLE
AND T0036  ; OPERATION.AUTO.CYCLE.SEQUENCE.STEP8.TIMER
SET H7.08  ; OPERATION.AUTO.CYCLE.SEQUENCE.STEP9
RSET H7.07  ; OPERATION.AUTO.CYCLE.SEQUENCE.STEP8
; rung 33: Step Timer
LD H7.07  ; OPERATION.AUTO.CYCLE.SEQUENCE.STEP8
TIM 0036 #15  ; OPERATION.AUTO.CYCLE.SEQUENCE.STEP8.TIMER
; rung 34
LD H7.08  ; OPERATION.AUTO.CYCLE.SEQUENCE.STEP9
AND H9.15  ; OPERATION.AUTO.CYCLE.STEP.ENABLE
AND T0037  ; OPERATION.AUTO.CYCLE.SEQUENCE.STEP9.TIMER
AND H20.08  ; OPERATION.LONG.AXIS.IN.POSITION.WINDOW.TOLERANCE
SET H7.09  ; OPERATION.AUTO.CYCLE.SEQUENCE.STEP10
RSET H7.08  ; OPERATION.AUTO.CYCLE.SEQUENCE.STEP9
; rung 35: Step Timer
LD H7.08  ; OPERATION.AUTO.CYCLE.SEQUENCE.STEP9
TIM 0037 #5  ; OPERATION.AUTO.CYCLE.SEQUENCE.STEP9.TIMER

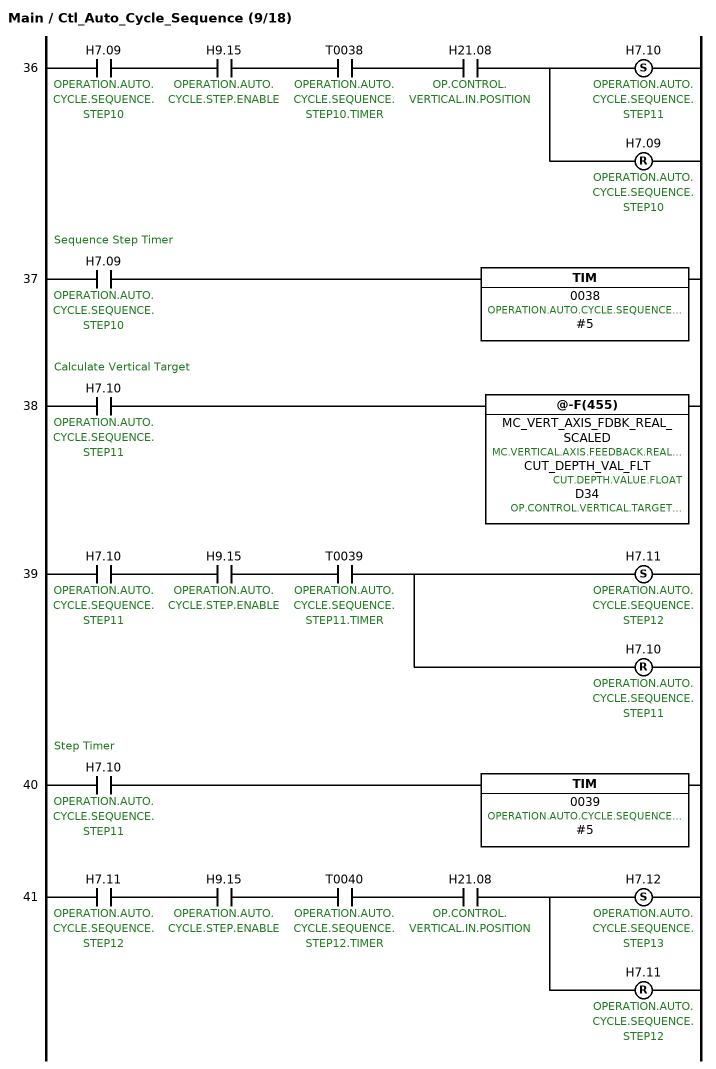
; rung 36
LD H7.09  ; OPERATION.AUTO.CYCLE.SEQUENCE.STEP10
AND H9.15  ; OPERATION.AUTO.CYCLE.STEP.ENABLE
AND T0038  ; OPERATION.AUTO.CYCLE.SEQUENCE.STEP10.TIMER
AND H21.08  ; OP.CONTROL.VERTICAL.IN.POSITION
SET H7.10  ; OPERATION.AUTO.CYCLE.SEQUENCE.STEP11
RSET H7.09  ; OPERATION.AUTO.CYCLE.SEQUENCE.STEP10
; rung 37: Sequence Step Timer
LD H7.09  ; OPERATION.AUTO.CYCLE.SEQUENCE.STEP10
TIM 0038 #5  ; OPERATION.AUTO.CYCLE.SEQUENCE.STEP10.TIMER
; rung 38: Calculate Vertical Target
LD H7.10  ; OPERATION.AUTO.CYCLE.SEQUENCE.STEP11
@-F(455) MC_VERT_AXIS_FDBK_REAL_SCALED CUT_DEPTH_VAL_FLT D34  ; MC.VERTICAL.AXIS.FEEDBACK.REAL.SCALED.INCH, CUT.DEPTH.VALUE.FLOAT, OP.CONTROL.VERTICAL.TARGET.SCALED
; rung 39
LD H7.10  ; OPERATION.AUTO.CYCLE.SEQUENCE.STEP11
AND H9.15  ; OPERATION.AUTO.CYCLE.STEP.ENABLE
AND T0039  ; OPERATION.AUTO.CYCLE.SEQUENCE.STEP11.TIMER
SET H7.11  ; OPERATION.AUTO.CYCLE.SEQUENCE.STEP12
RSET H7.10  ; OPERATION.AUTO.CYCLE.SEQUENCE.STEP11
; rung 40: Step Timer
LD H7.10  ; OPERATION.AUTO.CYCLE.SEQUENCE.STEP11
TIM 0039 #5  ; OPERATION.AUTO.CYCLE.SEQUENCE.STEP11.TIMER
; rung 41
LD H7.11  ; OPERATION.AUTO.CYCLE.SEQUENCE.STEP12
AND H9.15  ; OPERATION.AUTO.CYCLE.STEP.ENABLE
AND T0040  ; OPERATION.AUTO.CYCLE.SEQUENCE.STEP12.TIMER
AND H21.08  ; OP.CONTROL.VERTICAL.IN.POSITION
SET H7.12  ; OPERATION.AUTO.CYCLE.SEQUENCE.STEP13
RSET H7.11  ; OPERATION.AUTO.CYCLE.SEQUENCE.STEP12

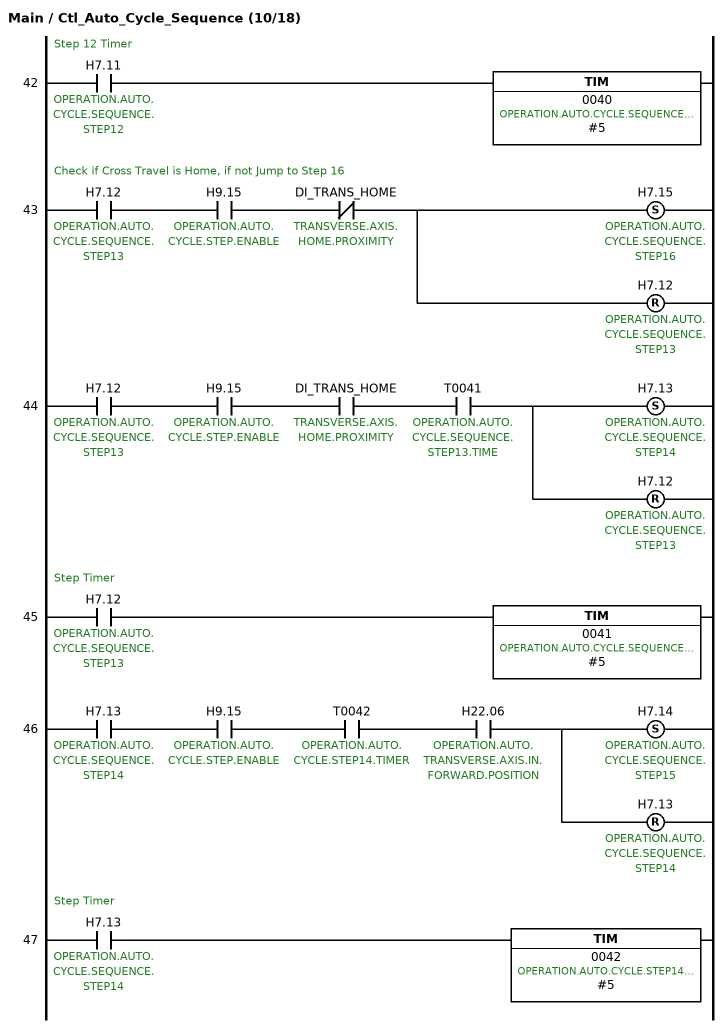
; rung 42: Step 12 Timer
LD H7.11  ; OPERATION.AUTO.CYCLE.SEQUENCE.STEP12
TIM 0040 #5  ; OPERATION.AUTO.CYCLE.SEQUENCE.STEP12.TIMER
; rung 43: Check if Cross Travel is Home, if not Jump to Step 16
LD H7.12  ; OPERATION.AUTO.CYCLE.SEQUENCE.STEP13
AND H9.15  ; OPERATION.AUTO.CYCLE.STEP.ENABLE
ANDNOT DI_TRANS_HOME  ; TRANSVERSE.AXIS.HOME.PROXIMITY
SET H7.15  ; OPERATION.AUTO.CYCLE.SEQUENCE.STEP16
RSET H7.12  ; OPERATION.AUTO.CYCLE.SEQUENCE.STEP13
; rung 44
LD H7.12  ; OPERATION.AUTO.CYCLE.SEQUENCE.STEP13
AND H9.15  ; OPERATION.AUTO.CYCLE.STEP.ENABLE
AND DI_TRANS_HOME  ; TRANSVERSE.AXIS.HOME.PROXIMITY
AND T0041  ; OPERATION.AUTO.CYCLE.SEQUENCE.STEP13.TIME
SET H7.13  ; OPERATION.AUTO.CYCLE.SEQUENCE.STEP14
RSET H7.12  ; OPERATION.AUTO.CYCLE.SEQUENCE.STEP13
; rung 45: Step Timer
LD H7.12  ; OPERATION.AUTO.CYCLE.SEQUENCE.STEP13
TIM 0041 #5  ; OPERATION.AUTO.CYCLE.SEQUENCE.STEP13.TIME
; rung 46
LD H7.13  ; OPERATION.AUTO.CYCLE.SEQUENCE.STEP14
AND H9.15  ; OPERATION.AUTO.CYCLE.STEP.ENABLE
AND T0042  ; OPERATION.AUTO.CYCLE.STEP14.TIMER
AND H22.06  ; OPERATION.AUTO.TRANSVERSE.AXIS.IN.FORWARD.POSITION
SET H7.14  ; OPERATION.AUTO.CYCLE.SEQUENCE.STEP15
RSET H7.13  ; OPERATION.AUTO.CYCLE.SEQUENCE.STEP14
; rung 47: Step Timer
LD H7.13  ; OPERATION.AUTO.CYCLE.SEQUENCE.STEP14
TIM 0042 #5  ; OPERATION.AUTO.CYCLE.STEP14.TIMER

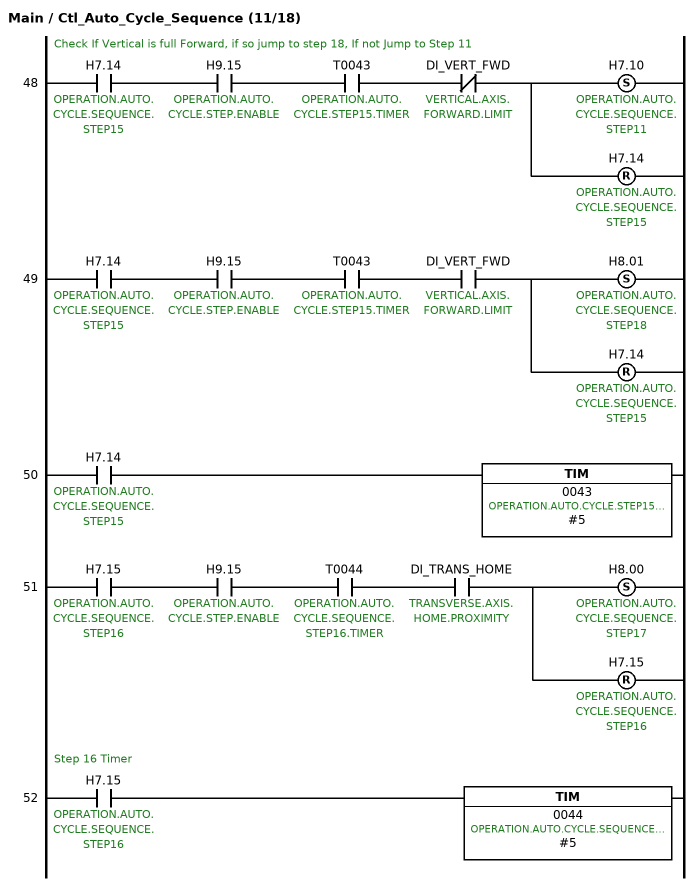
; rung 48: Check If Vertical is full Forward, if so jump to step 18, If not Jump to Step 11
LD H7.14  ; OPERATION.AUTO.CYCLE.SEQUENCE.STEP15
AND H9.15  ; OPERATION.AUTO.CYCLE.STEP.ENABLE
AND T0043  ; OPERATION.AUTO.CYCLE.STEP15.TIMER
ANDNOT DI_VERT_FWD  ; VERTICAL.AXIS.FORWARD.LIMIT
SET H7.10  ; OPERATION.AUTO.CYCLE.SEQUENCE.STEP11
RSET H7.14  ; OPERATION.AUTO.CYCLE.SEQUENCE.STEP15
; rung 49
LD H7.14  ; OPERATION.AUTO.CYCLE.SEQUENCE.STEP15
AND H9.15  ; OPERATION.AUTO.CYCLE.STEP.ENABLE
AND T0043  ; OPERATION.AUTO.CYCLE.STEP15.TIMER
AND DI_VERT_FWD  ; VERTICAL.AXIS.FORWARD.LIMIT
SET H8.01  ; OPERATION.AUTO.CYCLE.SEQUENCE.STEP18
RSET H7.14  ; OPERATION.AUTO.CYCLE.SEQUENCE.STEP15
; rung 50
LD H7.14  ; OPERATION.AUTO.CYCLE.SEQUENCE.STEP15
TIM 0043 #5  ; OPERATION.AUTO.CYCLE.STEP15.TIMER
; rung 51
LD H7.15  ; OPERATION.AUTO.CYCLE.SEQUENCE.STEP16
AND H9.15  ; OPERATION.AUTO.CYCLE.STEP.ENABLE
AND T0044  ; OPERATION.AUTO.CYCLE.SEQUENCE.STEP16.TIMER
AND DI_TRANS_HOME  ; TRANSVERSE.AXIS.HOME.PROXIMITY
SET H8.00  ; OPERATION.AUTO.CYCLE.SEQUENCE.STEP17
RSET H7.15  ; OPERATION.AUTO.CYCLE.SEQUENCE.STEP16
; rung 52: Step 16 Timer
LD H7.15  ; OPERATION.AUTO.CYCLE.SEQUENCE.STEP16
TIM 0044 #5  ; OPERATION.AUTO.CYCLE.SEQUENCE.STEP16.TIMER

